(* Logix 5000 project; controller reports 1756-L63 rev 20.11; software revision 20.04; part 45 of 52 *)

        [132].log_data[58].valid := 1, [132].log_data[59].time := 3600.0, [132].log_data[59].valid := 1, [132].log_data[60].valid := 1, [132].log_data[61].valid := 1, [132].log_data[62].valid := 1, [132].log_data[63].valid := 1, [132].log_data[64].valid := 1, [132].log_data[65].valid := 1, [132].log_data[66].valid := 1, [132].log_data[67].valid := 1, [132].log_data[68].valid := 1, [132].log_data[69].valid := 1, [132].log_data[70].valid := 1, [132].log_data[71].valid := 1, [132].log_data[72].valid := 1, [132].log_data[73].valid := 1, [132].log_data[74].valid := 1, [132].log_data[75].valid := 1, [132].log_data[76].valid := 1, [132].log_data[77].valid := 1, [132].log_data[78].valid := 1, [132].log_data[79].valid := 1, [132].log_data[80].valid := 1, [132].log_data[81].valid := 1, [132].log_data[82].valid := 1, [132].log_data[83].valid := 1, [132].log_data[84].valid := 1, [132].log_data[85].valid := 1, [132].log_data[86].valid := 1, [132].log_data[87].valid := 1, [132].log_data[88].valid := 1, [132].log_data[89].valid := 1, [132].log_data[90].valid := 1, [132].log_data[91].valid := 1, [132].log_data[92].valid := 1, [132].log_data[93].valid := 1, [132].log_data[94].valid := 1, [132].log_data[95].valid := 1, [132].log_data[96].valid := 1, [132].log_data[97].valid := 1, [132].log_data[98].valid := 1, [132].log_data[99].valid := 1, [132].log_data[100].valid := 1, [132].log_data[101].valid := 1, [132].log_data[102].valid := 1, [132].log_data[103].valid := 1, [132].log_data[104].valid := 1, [132].log_data[105].valid := 1, [132].log_data[106].valid := 1, [132].log_data[107].valid := 1, [132].log_data[108].valid := 1, [132].log_data[109].valid := 1, [132].log_data[110].valid := 1, [132].log_data[111].valid := 1, [132].log_data[112].valid := 1, [132].log_data[113].valid := 1, [132].log_data[114].valid := 1, [132].log_data[115].valid := 1, [132].log_data[116].valid := 1,
        [132].log_data[117].valid := 1, [132].log_data[118].valid := 1, [132].log_data[119].valid := 1, [132].log_data[120].valid := 1, [132].log_data[121].valid := 1, [132].log_data[122].valid := 1, [132].log_data[123].valid := 1, [132].log_data[124].valid := 1, [132].time.Year := 2023, [132].time.Month := 1, [132].time.Day := 18, [132].time.Hour := 15, [132].time.Minute := 59, [132].time.Second := 59, [133].log_data[0].min := 1.0, [133].log_data[0].max := 1.0, [133].log_data[0].total := 3600.0, [133].log_data[0].time := 3600.0, [133].log_data[0].valid := 1, [133].log_data[1].max := 1.0, [133].log_data[1].total := 561.5, [133].log_data[1].time := 3600.0, [133].log_data[1].maxminute := 34, [133].log_data[1].valid := 1, [133].log_data[2].max := 1.0, [133].log_data[2].total := 558.0, [133].log_data[2].time := 3600.0, [133].log_data[2].maxminute := 34, [133].log_data[2].valid := 1, [133].log_data[3].time := 3600.0, [133].log_data[3].valid := 1, [133].log_data[4].time := 3600.0, [133].log_data[4].valid := 1, [133].log_data[5].max := 1.0, [133].log_data[5].total := 252.0, [133].log_data[5].time := 3600.0, [133].log_data[5].maxminute := 36, [133].log_data[5].valid := 1, [133].log_data[6].time := 3600.0, [133].log_data[6].valid := 1, [133].log_data[7].time := 3600.0, [133].log_data[7].valid := 1, [133].log_data[8].time := 3600.0, [133].log_data[8].valid := 1, [133].log_data[9].time := 3600.0, [133].log_data[9].valid := 1, [133].log_data[10].min := 1.0, [133].log_data[10].max := 1.0, [133].log_data[10].total := 3600.0, [133].log_data[10].time := 3600.0, [133].log_data[10].valid := 1, [133].log_data[11].time := 3600.0, [133].log_data[11].valid := 1, [133].log_data[12].min := 1.0, [133].log_data[12].max := 1.0, [133].log_data[12].total := 3600.0, [133].log_data[12].time := 3600.0, [133].log_data[12].valid := 1, [133].log_data[13].min := 1.0, [133].log_data[13].max := 1.0,
        [133].log_data[13].total := 3600.0, [133].log_data[13].time := 3600.0, [133].log_data[13].valid := 1, [133].log_data[14].time := 3600.0, [133].log_data[14].valid := 1, [133].log_data[15].time := 3600.0, [133].log_data[15].valid := 1, [133].log_data[16].time := 3600.0, [133].log_data[16].valid := 1, [133].log_data[17].min := 1.0, [133].log_data[17].max := 1.0, [133].log_data[17].total := 3600.0, [133].log_data[17].time := 3600.0, [133].log_data[17].valid := 1, [133].log_data[18].time := 3600.0, [133].log_data[18].valid := 1, [133].log_data[19].time := 3600.0, [133].log_data[19].valid := 1, [133].log_data[20].time := 3600.0, [133].log_data[20].valid := 1, [133].log_data[21].min := 1.0, [133].log_data[21].max := 1.0, [133].log_data[21].total := 3600.0, [133].log_data[21].time := 3600.0, [133].log_data[21].valid := 1, [133].log_data[22].time := 3600.0, [133].log_data[22].valid := 1, [133].log_data[23].time := 3600.0, [133].log_data[23].valid := 1, [133].log_data[24].time := 3600.0, [133].log_data[24].valid := 1, [133].log_data[25].time := 3600.0, [133].log_data[25].valid := 1, [133].log_data[26].time := 3600.0, [133].log_data[26].valid := 1, [133].log_data[27].time := 3600.0, [133].log_data[27].valid := 1, [133].log_data[28].time := 3600.0, [133].log_data[28].valid := 1, [133].log_data[29].min := 1.0, [133].log_data[29].max := 1.0, [133].log_data[29].total := 3600.0, [133].log_data[29].time := 3600.0, [133].log_data[29].valid := 1, [133].log_data[30].min := 1.0, [133].log_data[30].max := 1.0, [133].log_data[30].total := 3600.0, [133].log_data[30].time := 3600.0, [133].log_data[30].valid := 1, [133].log_data[31].time := 3600.0, [133].log_data[31].valid := 1, [133].log_data[32].time := 3600.0, [133].log_data[32].valid := 1, [133].log_data[33].time := 3600.0, [133].log_data[33].valid := 1, [133].log_data[34].time := 3600.0, [133].log_data[34].valid := 1, [133].log_data[35].time := 3600.0, [133].log_data[35].valid := 1, [133].log_data[36].time := 3600.0,
        [133].log_data[36].valid := 1, [133].log_data[37].max := 7.5544033, [133].log_data[37].total := 3699.229, [133].log_data[37].time := 3600.0, [133].log_data[37].maxminute := 36, [133].log_data[37].valid := 1, [133].log_data[38].time := 3600.0, [133].log_data[38].valid := 1, [133].log_data[39].min := 0.99541295, [133].log_data[39].max := 1.0215589, [133].log_data[39].total := 3606.4697, [133].log_data[39].time := 3600.0, [133].log_data[39].minminute := 45, [133].log_data[39].maxminute := 41, [133].log_data[39].valid := 1, [133].log_data[40].min := 7.5885, [133].log_data[40].max := 7.6244993, [133].log_data[40].total := 27393.127, [133].log_data[40].time := 3600.0, [133].log_data[40].minminute := 44, [133].log_data[40].maxminute := 51, [133].log_data[40].valid := 1, [133].log_data[41].min := 0.022343751, [133].log_data[41].max := 0.022932617, [133].log_data[41].total := 81.647255, [133].log_data[41].time := 3600.0, [133].log_data[41].minminute := 10, [133].log_data[41].valid := 1, [133].log_data[42].min := 2.291407, [133].log_data[42].max := 2.2958827, [133].log_data[42].total := 8257.927, [133].log_data[42].time := 3600.0, [133].log_data[42].minminute := 49, [133].log_data[42].maxminute := 6, [133].log_data[42].valid := 1, [133].log_data[43].min := -0.26000214, [133].log_data[43].max := -0.23999786, [133].log_data[43].total := -932.50854, [133].log_data[43].time := 3600.0, [133].log_data[43].valid := 1, [133].log_data[44].min := -0.30000305, [133].log_data[44].max := -0.27999878, [133].log_data[44].total := -1009.3977, [133].log_data[44].time := 3600.0, [133].log_data[44].valid := 1, [133].log_data[45].time := 3600.0, [133].log_data[45].valid := 1, [133].log_data[46].time := 3600.0, [133].log_data[46].valid := 1, [133].log_data[47].time := 3600.0, [133].log_data[47].valid := 1, [133].log_data[48].min := 6.7547326, [133].log_data[48].max := 6.977601, [133].log_data[48].total := 24541.125, [133].log_data[48].time := 3600.0, [133].log_data[48].maxminute := 43, [133].log_data[48].valid := 1, [133].log_data[49].min := 6.734528, [133].log_data[49].max := 9.605879, [133].log_data[49].total := 31908.559,
        [133].log_data[49].time := 3600.0, [133].log_data[49].minminute := 59, [133].log_data[49].maxminute := 37, [133].log_data[49].valid := 1, [133].log_data[50].min := 2.00227, [133].log_data[50].max := 2.1381822, [133].log_data[50].total := 7381.451, [133].log_data[50].time := 3600.0, [133].log_data[50].minminute := 11, [133].log_data[50].maxminute := 57, [133].log_data[50].valid := 1, [133].log_data[51].time := 3600.0, [133].log_data[51].valid := 1, [133].log_data[52].min := -1.6200027, [133].log_data[52].max := -1.4800034, [133].log_data[52].total := -5649.4478, [133].log_data[52].time := 3600.0, [133].log_data[52].minminute := 4, [133].log_data[52].maxminute := 31, [133].log_data[52].valid := 1, [133].log_data[53].min := -1.5800018, [133].log_data[53].max := -1.4599991, [133].log_data[53].total := -5378.804, [133].log_data[53].time := 3600.0, [133].log_data[53].minminute := 12, [133].log_data[53].maxminute := 1, [133].log_data[53].valid := 1, [133].log_data[54].time := 3600.0, [133].log_data[54].valid := 1, [133].log_data[55].time := 3600.0, [133].log_data[55].valid := 1, [133].log_data[56].min := 0.15898935, [133].log_data[56].max := 0.15938194, [133].log_data[56].total := 573.0084, [133].log_data[56].time := 3600.0, [133].log_data[56].minminute := 59, [133].log_data[56].maxminute := 7, [133].log_data[56].valid := 1, [133].log_data[57].min := 0.20103496, [133].log_data[57].max := 0.20142753, [133].log_data[57].total := 724.2275, [133].log_data[57].time := 3600.0, [133].log_data[57].minminute := 2, [133].log_data[57].maxminute := 41, [133].log_data[57].valid := 1, [133].log_data[58].time := 3600.0, [133].log_data[58].valid := 1, [133].log_data[59].time := 3600.0, [133].log_data[59].valid := 1, [133].log_data[60].valid := 1, [133].log_data[61].valid := 1, [133].log_data[62].valid := 1, [133].log_data[63].valid := 1, [133].log_data[64].valid := 1, [133].log_data[65].valid := 1, [133].log_data[66].valid := 1, [133].log_data[67].valid := 1, [133].log_data[68].valid := 1, [133].log_data[69].valid := 1, [133].log_data[70].valid := 1,
        [133].log_data[71].valid := 1, [133].log_data[72].valid := 1, [133].log_data[73].valid := 1, [133].log_data[74].valid := 1, [133].log_data[75].valid := 1, [133].log_data[76].valid := 1, [133].log_data[77].valid := 1, [133].log_data[78].valid := 1, [133].log_data[79].valid := 1, [133].log_data[80].valid := 1, [133].log_data[81].valid := 1, [133].log_data[82].valid := 1, [133].log_data[83].valid := 1, [133].log_data[84].valid := 1, [133].log_data[85].valid := 1, [133].log_data[86].valid := 1, [133].log_data[87].valid := 1, [133].log_data[88].valid := 1, [133].log_data[89].valid := 1, [133].log_data[90].valid := 1, [133].log_data[91].valid := 1, [133].log_data[92].valid := 1, [133].log_data[93].valid := 1, [133].log_data[94].valid := 1, [133].log_data[95].valid := 1, [133].log_data[96].valid := 1, [133].log_data[97].valid := 1, [133].log_data[98].valid := 1, [133].log_data[99].valid := 1, [133].log_data[100].valid := 1, [133].log_data[101].valid := 1, [133].log_data[102].valid := 1, [133].log_data[103].valid := 1, [133].log_data[104].valid := 1, [133].log_data[105].valid := 1, [133].log_data[106].valid := 1, [133].log_data[107].valid := 1, [133].log_data[108].valid := 1, [133].log_data[109].valid := 1, [133].log_data[110].valid := 1, [133].log_data[111].valid := 1, [133].log_data[112].valid := 1, [133].log_data[113].valid := 1, [133].log_data[114].valid := 1, [133].log_data[115].valid := 1, [133].log_data[116].valid := 1, [133].log_data[117].valid := 1, [133].log_data[118].valid := 1, [133].log_data[119].valid := 1, [133].log_data[120].valid := 1, [133].log_data[121].valid := 1, [133].log_data[122].valid := 1, [133].log_data[123].valid := 1, [133].log_data[124].valid := 1, [133].time.Year := 2023, [133].time.Month := 1, [133].time.Day := 18, [133].time.Hour := 16, [133].time.Minute := 59, [133].time.Second := 59,
        [134].log_data[0].min := 1.0, [134].log_data[0].max := 1.0, [134].log_data[0].total := 3600.0, [134].log_data[0].time := 3600.0, [134].log_data[0].valid := 1, [134].log_data[1].max := 1.0, [134].log_data[1].total := 524.749, [134].log_data[1].time := 3600.0, [134].log_data[1].maxminute := 51, [134].log_data[1].valid := 1, [134].log_data[2].max := 1.0, [134].log_data[2].total := 521.249, [134].log_data[2].time := 3600.0, [134].log_data[2].maxminute := 51, [134].log_data[2].valid := 1, [134].log_data[3].time := 3600.0, [134].log_data[3].valid := 1, [134].log_data[4].time := 3600.0, [134].log_data[4].valid := 1, [134].log_data[5].max := 1.0, [134].log_data[5].total := 224.249, [134].log_data[5].time := 3600.0, [134].log_data[5].maxminute := 53, [134].log_data[5].valid := 1, [134].log_data[6].time := 3600.0, [134].log_data[6].valid := 1, [134].log_data[7].time := 3600.0, [134].log_data[7].valid := 1, [134].log_data[8].max := 1.0, [134].log_data[8].total := 337.749, [134].log_data[8].time := 3600.0, [134].log_data[8].maxminute := 54, [134].log_data[8].valid := 1, [134].log_data[9].max := 1.0, [134].log_data[9].total := 334.249, [134].log_data[9].time := 3600.0, [134].log_data[9].maxminute := 54, [134].log_data[9].valid := 1, [134].log_data[10].min := 1.0, [134].log_data[10].max := 1.0, [134].log_data[10].total := 3600.0, [134].log_data[10].time := 3600.0, [134].log_data[10].valid := 1, [134].log_data[11].time := 3600.0, [134].log_data[11].valid := 1, [134].log_data[12].min := 1.0, [134].log_data[12].max := 1.0, [134].log_data[12].total := 3600.0, [134].log_data[12].time := 3600.0, [134].log_data[12].valid := 1, [134].log_data[13].min := 1.0, [134].log_data[13].max := 1.0, [134].log_data[13].total := 3600.0, [134].log_data[13].time := 3600.0, [134].log_data[13].valid := 1, [134].log_data[14].time := 3600.0, [134].log_data[14].valid := 1, [134].log_data[15].time := 3600.0, [134].log_data[15].valid := 1, [134].log_data[16].time := 3600.0,
        [134].log_data[16].valid := 1, [134].log_data[17].min := 1.0, [134].log_data[17].max := 1.0, [134].log_data[17].total := 3600.0, [134].log_data[17].time := 3600.0, [134].log_data[17].valid := 1, [134].log_data[18].time := 3600.0, [134].log_data[18].valid := 1, [134].log_data[19].time := 3600.0, [134].log_data[19].valid := 1, [134].log_data[20].time := 3600.0, [134].log_data[20].valid := 1, [134].log_data[21].min := 1.0, [134].log_data[21].max := 1.0, [134].log_data[21].total := 3600.0, [134].log_data[21].time := 3600.0, [134].log_data[21].valid := 1, [134].log_data[22].time := 3600.0, [134].log_data[22].valid := 1, [134].log_data[23].time := 3600.0, [134].log_data[23].valid := 1, [134].log_data[24].time := 3600.0, [134].log_data[24].valid := 1, [134].log_data[25].time := 3600.0, [134].log_data[25].valid := 1, [134].log_data[26].time := 3600.0, [134].log_data[26].valid := 1, [134].log_data[27].time := 3600.0, [134].log_data[27].valid := 1, [134].log_data[28].time := 3600.0, [134].log_data[28].valid := 1, [134].log_data[29].min := 1.0, [134].log_data[29].max := 1.0, [134].log_data[29].total := 3600.0, [134].log_data[29].time := 3600.0, [134].log_data[29].valid := 1, [134].log_data[30].min := 1.0, [134].log_data[30].max := 1.0, [134].log_data[30].total := 3600.0, [134].log_data[30].time := 3600.0, [134].log_data[30].valid := 1, [134].log_data[31].max := 1.0, [134].log_data[31].total := 57.249, [134].log_data[31].time := 3600.0, [134].log_data[31].maxminute := 54, [134].log_data[31].valid := 1, [134].log_data[32].max := 1.0, [134].log_data[32].total := 185.249, [134].log_data[32].time := 3600.0, [134].log_data[32].maxminute := 56, [134].log_data[32].valid := 1, [134].log_data[33].time := 3600.0, [134].log_data[33].valid := 1, [134].log_data[34].time := 3600.0, [134].log_data[34].valid := 1, [134].log_data[35].time := 3600.0, [134].log_data[35].valid := 1, [134].log_data[36].max := 1.0, [134].log_data[36].total := 327.249, [134].log_data[36].time := 3600.0,
        [134].log_data[36].maxminute := 54, [134].log_data[36].valid := 1, [134].log_data[37].max := 9.523992, [134].log_data[37].total := 3687.952, [134].log_data[37].time := 3600.0, [134].log_data[37].maxminute := 53, [134].log_data[37].valid := 1, [134].log_data[38].time := 3600.0, [134].log_data[38].valid := 1, [134].log_data[39].min := 0.99423516, [134].log_data[39].max := 1.0213233, [134].log_data[39].total := 3603.442, [134].log_data[39].time := 3600.0, [134].log_data[39].minminute := 13, [134].log_data[39].maxminute := 58, [134].log_data[39].valid := 1, [134].log_data[40].min := 7.592622, [134].log_data[40].max := 7.6244993, [134].log_data[40].total := 27393.01, [134].log_data[40].time := 3600.0, [134].log_data[40].minminute := 1, [134].log_data[40].maxminute := 10, [134].log_data[40].valid := 1, [134].log_data[41].min := 0.022343751, [134].log_data[41].max := 0.022932617, [134].log_data[41].total := 81.438286, [134].log_data[41].time := 3600.0, [134].log_data[41].minminute := 1, [134].log_data[41].maxminute := 15, [134].log_data[41].valid := 1, [134].log_data[42].min := 2.2912893, [134].log_data[42].max := 2.296118, [134].log_data[42].total := 8257.677, [134].log_data[42].time := 3600.0, [134].log_data[42].minminute := 38, [134].log_data[42].maxminute := 18, [134].log_data[42].valid := 1, [134].log_data[43].min := -0.26000214, [134].log_data[43].max := -0.23999786, [134].log_data[43].total := -926.4218, [134].log_data[43].time := 3600.0, [134].log_data[43].maxminute := 1, [134].log_data[43].valid := 1, [134].log_data[44].min := -0.30000305, [134].log_data[44].max := -0.27999878, [134].log_data[44].total := -1008.3122, [134].log_data[44].time := 3600.0, [134].log_data[44].valid := 1, [134].log_data[45].time := 3600.0, [134].log_data[45].valid := 1, [134].log_data[46].time := 3600.0, [134].log_data[46].valid := 1, [134].log_data[47].time := 3600.0, [134].log_data[47].valid := 1, [134].log_data[48].min := 6.618977, [134].log_data[48].max := 6.854762, [134].log_data[48].total := 24051.516, [134].log_data[48].time := 3600.0, [134].log_data[48].minminute := 28, [134].log_data[48].maxminute := 59,
        [134].log_data[48].valid := 1, [134].log_data[49].min := 6.092655, [134].log_data[49].max := 8.969305, [134].log_data[49].total := 25809.742, [134].log_data[49].time := 3600.0, [134].log_data[49].minminute := 16, [134].log_data[49].maxminute := 54, [134].log_data[49].valid := 1, [134].log_data[50].min := 2.0787058, [134].log_data[50].max := 2.1524327, [134].log_data[50].total := 7686.3364, [134].log_data[50].time := 3600.0, [134].log_data[50].minminute := 58, [134].log_data[50].maxminute := 54, [134].log_data[50].valid := 1, [134].log_data[51].time := 3600.0, [134].log_data[51].valid := 1, [134].log_data[52].min := -4.119995, [134].log_data[52].max := 0.13999939, [134].log_data[52].total := -5775.382, [134].log_data[52].time := 3600.0, [134].log_data[52].minminute := 54, [134].log_data[52].maxminute := 56, [134].log_data[52].valid := 1, [134].log_data[53].min := -4.079994, [134].log_data[53].max := -1.4599991, [134].log_data[53].total := -5722.698, [134].log_data[53].time := 3600.0, [134].log_data[53].minminute := 54, [134].log_data[53].valid := 1, [134].log_data[54].max := 0.513, [134].log_data[54].total := 92.831985, [134].log_data[54].time := 3600.0, [134].log_data[54].maxminute := 57, [134].log_data[54].valid := 1, [134].log_data[55].max := 0.526, [134].log_data[55].total := 128.63133, [134].log_data[55].time := 3600.0, [134].log_data[55].maxminute := 54, [134].log_data[55].valid := 1, [134].log_data[56].min := 0.15898935, [134].log_data[56].max := 0.15942119, [134].log_data[56].total := 572.9697, [134].log_data[56].time := 3600.0, [134].log_data[56].minminute := 45, [134].log_data[56].maxminute := 38, [134].log_data[56].valid := 1, [134].log_data[57].min := 0.20103496, [134].log_data[57].max := 0.20142753, [134].log_data[57].total := 724.2705, [134].log_data[57].time := 3600.0, [134].log_data[57].maxminute := 36, [134].log_data[57].valid := 1, [134].log_data[58].time := 3600.0, [134].log_data[58].valid := 1, [134].log_data[59].time := 3600.0, [134].log_data[59].valid := 1, [134].log_data[60].valid := 1, [134].log_data[61].valid := 1, [134].log_data[62].valid := 1,
        [134].log_data[63].valid := 1, [134].log_data[64].valid := 1, [134].log_data[65].valid := 1, [134].log_data[66].valid := 1, [134].log_data[67].valid := 1, [134].log_data[68].valid := 1, [134].log_data[69].valid := 1, [134].log_data[70].valid := 1, [134].log_data[71].valid := 1, [134].log_data[72].valid := 1, [134].log_data[73].valid := 1, [134].log_data[74].valid := 1, [134].log_data[75].valid := 1, [134].log_data[76].valid := 1, [134].log_data[77].valid := 1, [134].log_data[78].valid := 1, [134].log_data[79].valid := 1, [134].log_data[80].valid := 1, [134].log_data[81].valid := 1, [134].log_data[82].valid := 1, [134].log_data[83].valid := 1, [134].log_data[84].valid := 1, [134].log_data[85].valid := 1, [134].log_data[86].valid := 1, [134].log_data[87].valid := 1, [134].log_data[88].valid := 1, [134].log_data[89].valid := 1, [134].log_data[90].valid := 1, [134].log_data[91].valid := 1, [134].log_data[92].valid := 1, [134].log_data[93].valid := 1, [134].log_data[94].valid := 1, [134].log_data[95].valid := 1, [134].log_data[96].valid := 1, [134].log_data[97].valid := 1, [134].log_data[98].valid := 1, [134].log_data[99].valid := 1, [134].log_data[100].valid := 1, [134].log_data[101].valid := 1, [134].log_data[102].valid := 1, [134].log_data[103].valid := 1, [134].log_data[104].valid := 1, [134].log_data[105].valid := 1, [134].log_data[106].valid := 1, [134].log_data[107].valid := 1, [134].log_data[108].valid := 1, [134].log_data[109].valid := 1, [134].log_data[110].valid := 1, [134].log_data[111].valid := 1, [134].log_data[112].valid := 1, [134].log_data[113].valid := 1, [134].log_data[114].valid := 1, [134].log_data[115].valid := 1, [134].log_data[116].valid := 1, [134].log_data[117].valid := 1, [134].log_data[118].valid := 1, [134].log_data[119].valid := 1, [134].log_data[120].valid := 1, [134].log_data[121].valid := 1, [134].log_data[122].valid := 1,
        [134].log_data[123].valid := 1, [134].log_data[124].valid := 1, [134].time.Year := 2023, [134].time.Month := 1, [134].time.Day := 18, [134].time.Hour := 17, [134].time.Minute := 59, [134].time.Second := 59, [135].log_data[0].min := 1.0, [135].log_data[0].max := 1.0, [135].log_data[0].total := 3600.0, [135].log_data[0].time := 3600.0, [135].log_data[0].valid := 1, [135].log_data[1].max := 1.0, [135].log_data[1].total := 41.751, [135].log_data[1].time := 3600.0, [135].log_data[1].valid := 1, [135].log_data[2].max := 1.0, [135].log_data[2].total := 41.751, [135].log_data[2].time := 3600.0, [135].log_data[2].valid := 1, [135].log_data[3].time := 3600.0, [135].log_data[3].valid := 1, [135].log_data[4].time := 3600.0, [135].log_data[4].valid := 1, [135].log_data[5].max := 1.0, [135].log_data[5].total := 18.751, [135].log_data[5].time := 3600.0, [135].log_data[5].valid := 1, [135].log_data[6].time := 3600.0, [135].log_data[6].valid := 1, [135].log_data[7].time := 3600.0, [135].log_data[7].valid := 1, [135].log_data[8].min := 1.0, [135].log_data[8].max := 1.0, [135].log_data[8].total := 3600.0, [135].log_data[8].time := 3600.0, [135].log_data[8].valid := 1, [135].log_data[9].min := 1.0, [135].log_data[9].max := 1.0, [135].log_data[9].total := 3600.0, [135].log_data[9].time := 3600.0, [135].log_data[9].valid := 1, [135].log_data[10].min := 1.0, [135].log_data[10].max := 1.0, [135].log_data[10].total := 3600.0, [135].log_data[10].time := 3600.0, [135].log_data[10].valid := 1, [135].log_data[11].time := 3600.0, [135].log_data[11].valid := 1, [135].log_data[12].min := 1.0, [135].log_data[12].max := 1.0, [135].log_data[12].total := 3600.0, [135].log_data[12].time := 3600.0, [135].log_data[12].valid := 1, [135].log_data[13].min := 1.0, [135].log_data[13].max := 1.0, [135].log_data[13].total := 3600.0, [135].log_data[13].time := 3600.0, [135].log_data[13].valid := 1,
        [135].log_data[14].time := 3600.0, [135].log_data[14].valid := 1, [135].log_data[15].time := 3600.0, [135].log_data[15].valid := 1, [135].log_data[16].time := 3600.0, [135].log_data[16].valid := 1, [135].log_data[17].min := 1.0, [135].log_data[17].max := 1.0, [135].log_data[17].total := 3600.0, [135].log_data[17].time := 3600.0, [135].log_data[17].valid := 1, [135].log_data[18].time := 3600.0, [135].log_data[18].valid := 1, [135].log_data[19].time := 3600.0, [135].log_data[19].valid := 1, [135].log_data[20].time := 3600.0, [135].log_data[20].valid := 1, [135].log_data[21].min := 1.0, [135].log_data[21].max := 1.0, [135].log_data[21].total := 3600.0, [135].log_data[21].time := 3600.0, [135].log_data[21].valid := 1, [135].log_data[22].time := 3600.0, [135].log_data[22].valid := 1, [135].log_data[23].time := 3600.0, [135].log_data[23].valid := 1, [135].log_data[24].time := 3600.0, [135].log_data[24].valid := 1, [135].log_data[25].time := 3600.0, [135].log_data[25].valid := 1, [135].log_data[26].time := 3600.0, [135].log_data[26].valid := 1, [135].log_data[27].time := 3600.0, [135].log_data[27].valid := 1, [135].log_data[28].time := 3600.0, [135].log_data[28].valid := 1, [135].log_data[29].min := 1.0, [135].log_data[29].max := 1.0, [135].log_data[29].total := 3600.0, [135].log_data[29].time := 3600.0, [135].log_data[29].valid := 1, [135].log_data[30].min := 1.0, [135].log_data[30].max := 1.0, [135].log_data[30].total := 3600.0, [135].log_data[30].time := 3600.0, [135].log_data[30].valid := 1, [135].log_data[31].max := 1.0, [135].log_data[31].total := 1629.998, [135].log_data[31].time := 3600.0, [135].log_data[31].maxminute := 7, [135].log_data[31].valid := 1, [135].log_data[32].max := 1.0, [135].log_data[32].total := 1444.498, [135].log_data[32].time := 3600.0, [135].log_data[32].minminute := 5, [135].log_data[32].valid := 1, [135].log_data[33].time := 3600.0, [135].log_data[33].valid := 1, [135].log_data[34].time := 3600.0, [135].log_data[34].valid := 1,
        [135].log_data[35].max := 1.0, [135].log_data[35].total := 1629.498, [135].log_data[35].time := 3600.0, [135].log_data[35].maxminute := 2, [135].log_data[35].valid := 1, [135].log_data[36].max := 1.0, [135].log_data[36].total := 1440.998, [135].log_data[36].time := 3600.0, [135].log_data[36].minminute := 1, [135].log_data[36].valid := 1, [135].log_data[37].time := 3600.0, [135].log_data[37].valid := 1, [135].log_data[38].time := 3600.0, [135].log_data[38].valid := 1, [135].log_data[39].min := 0.99623734, [135].log_data[39].max := 1.0076615, [135].log_data[39].total := 3603.6245, [135].log_data[39].time := 3600.0, [135].log_data[39].minminute := 43, [135].log_data[39].valid := 1, [135].log_data[40].min := 7.586851, [135].log_data[40].max := 7.620378, [135].log_data[40].total := 27389.994, [135].log_data[40].time := 3600.0, [135].log_data[40].minminute := 28, [135].log_data[40].maxminute := 40, [135].log_data[40].valid := 1, [135].log_data[41].min := 0.022343751, [135].log_data[41].max := 0.022932617, [135].log_data[41].total := 81.52236, [135].log_data[41].time := 3600.0, [135].log_data[41].minminute := 4, [135].log_data[41].maxminute := 13, [135].log_data[41].valid := 1, [135].log_data[42].min := 2.290936, [135].log_data[42].max := 2.2957647, [135].log_data[42].total := 8257.714, [135].log_data[42].time := 3600.0, [135].log_data[42].minminute := 10, [135].log_data[42].maxminute := 5, [135].log_data[42].valid := 1, [135].log_data[43].min := -0.26000214, [135].log_data[43].max := -0.23999786, [135].log_data[43].total := -934.87366, [135].log_data[43].time := 3600.0, [135].log_data[43].valid := 1, [135].log_data[44].min := -0.30000305, [135].log_data[44].max := -0.27999878, [135].log_data[44].total := -1016.6125, [135].log_data[44].time := 3600.0, [135].log_data[44].valid := 1, [135].log_data[45].time := 3600.0, [135].log_data[45].valid := 1, [135].log_data[46].time := 3600.0, [135].log_data[46].valid := 1, [135].log_data[47].time := 3600.0, [135].log_data[47].valid := 1, [135].log_data[48].min := 6.677511, [135].log_data[48].max := 6.8819685, [135].log_data[48].total := 24228.434,
        [135].log_data[48].time := 3600.0, [135].log_data[48].minminute := 26, [135].log_data[48].valid := 1, [135].log_data[49].min := 6.88842, [135].log_data[49].max := 9.422542, [135].log_data[49].total := 28967.625, [135].log_data[49].time := 3600.0, [135].log_data[49].minminute := 21, [135].log_data[49].maxminute := 59, [135].log_data[49].valid := 1, [135].log_data[50].min := 2.059273, [135].log_data[50].max := 2.1438353, [135].log_data[50].total := 7571.9165, [135].log_data[50].time := 3600.0, [135].log_data[50].minminute := 59, [135].log_data[50].valid := 1, [135].log_data[51].time := 3600.0, [135].log_data[51].valid := 1, [135].log_data[52].min := -2.7600021, [135].log_data[52].max := 0.13999939, [135].log_data[52].total := -7516.524, [135].log_data[52].time := 3600.0, [135].log_data[52].minminute := 39, [135].log_data[52].maxminute := 6, [135].log_data[52].valid := 1, [135].log_data[53].min := -2.4400024, [135].log_data[53].max := 0.3600006, [135].log_data[53].total := -6614.5444, [135].log_data[53].time := 3600.0, [135].log_data[53].minminute := 46, [135].log_data[53].maxminute := 12, [135].log_data[53].valid := 1, [135].log_data[54].max := 0.5195, [135].log_data[54].total := 1221.1208, [135].log_data[54].time := 3600.0, [135].log_data[54].minminute := 5, [135].log_data[54].maxminute := 49, [135].log_data[54].valid := 1, [135].log_data[55].max := 0.557, [135].log_data[55].total := 1217.2502, [135].log_data[55].time := 3600.0, [135].log_data[55].minminute := 1, [135].log_data[55].maxminute := 2, [135].log_data[55].valid := 1, [135].log_data[56].min := 0.15898935, [135].log_data[56].max := 0.15938194, [135].log_data[56].total := 572.84296, [135].log_data[56].time := 3600.0, [135].log_data[56].minminute := 9, [135].log_data[56].maxminute := 37, [135].log_data[56].valid := 1, [135].log_data[57].min := 0.20095645, [135].log_data[57].max := 0.20138828, [135].log_data[57].total := 724.062, [135].log_data[57].time := 3600.0, [135].log_data[57].minminute := 19, [135].log_data[57].maxminute := 3, [135].log_data[57].valid := 1, [135].log_data[58].time := 3600.0, [135].log_data[58].valid := 1,
        [135].log_data[59].time := 3600.0, [135].log_data[59].valid := 1, [135].log_data[60].valid := 1, [135].log_data[61].valid := 1, [135].log_data[62].valid := 1, [135].log_data[63].valid := 1, [135].log_data[64].valid := 1, [135].log_data[65].valid := 1, [135].log_data[66].valid := 1, [135].log_data[67].valid := 1, [135].log_data[68].valid := 1, [135].log_data[69].valid := 1, [135].log_data[70].valid := 1, [135].log_data[71].valid := 1, [135].log_data[72].valid := 1, [135].log_data[73].valid := 1, [135].log_data[74].valid := 1, [135].log_data[75].valid := 1, [135].log_data[76].valid := 1, [135].log_data[77].valid := 1, [135].log_data[78].valid := 1, [135].log_data[79].valid := 1, [135].log_data[80].valid := 1, [135].log_data[81].valid := 1, [135].log_data[82].valid := 1, [135].log_data[83].valid := 1, [135].log_data[84].valid := 1, [135].log_data[85].valid := 1, [135].log_data[86].valid := 1, [135].log_data[87].valid := 1, [135].log_data[88].valid := 1, [135].log_data[89].valid := 1, [135].log_data[90].valid := 1, [135].log_data[91].valid := 1, [135].log_data[92].valid := 1, [135].log_data[93].valid := 1, [135].log_data[94].valid := 1, [135].log_data[95].valid := 1, [135].log_data[96].valid := 1, [135].log_data[97].valid := 1, [135].log_data[98].valid := 1, [135].log_data[99].valid := 1, [135].log_data[100].valid := 1, [135].log_data[101].valid := 1, [135].log_data[102].valid := 1, [135].log_data[103].valid := 1, [135].log_data[104].valid := 1, [135].log_data[105].valid := 1, [135].log_data[106].valid := 1, [135].log_data[107].valid := 1, [135].log_data[108].valid := 1, [135].log_data[109].valid := 1, [135].log_data[110].valid := 1, [135].log_data[111].valid := 1, [135].log_data[112].valid := 1, [135].log_data[113].valid := 1, [135].log_data[114].valid := 1, [135].log_data[115].valid := 1, [135].log_data[116].valid := 1, [135].log_data[117].valid := 1,
        [135].log_data[118].valid := 1, [135].log_data[119].valid := 1, [135].log_data[120].valid := 1, [135].log_data[121].valid := 1, [135].log_data[122].valid := 1, [135].log_data[123].valid := 1, [135].log_data[124].valid := 1, [135].time.Year := 2023, [135].time.Month := 1, [135].time.Day := 18, [135].time.Hour := 18, [135].time.Minute := 59, [135].time.Second := 59, [136].log_data[0].min := 1.0, [136].log_data[0].max := 1.0, [136].log_data[0].total := 3600.0, [136].log_data[0].time := 3600.0, [136].log_data[0].valid := 1, [136].log_data[1].max := 1.0, [136].log_data[1].total := 544.0, [136].log_data[1].time := 3600.0, [136].log_data[1].maxminute := 22, [136].log_data[1].valid := 1, [136].log_data[2].max := 1.0, [136].log_data[2].total := 540.5, [136].log_data[2].time := 3600.0, [136].log_data[2].maxminute := 22, [136].log_data[2].valid := 1, [136].log_data[3].time := 3600.0, [136].log_data[3].valid := 1, [136].log_data[4].time := 3600.0, [136].log_data[4].valid := 1, [136].log_data[5].max := 1.0, [136].log_data[5].total := 246.0, [136].log_data[5].time := 3600.0, [136].log_data[5].maxminute := 25, [136].log_data[5].valid := 1, [136].log_data[6].time := 3600.0, [136].log_data[6].valid := 1, [136].log_data[7].time := 3600.0, [136].log_data[7].valid := 1, [136].log_data[8].min := 1.0, [136].log_data[8].max := 1.0, [136].log_data[8].total := 3600.0, [136].log_data[8].time := 3600.0, [136].log_data[8].valid := 1, [136].log_data[9].min := 1.0, [136].log_data[9].max := 1.0, [136].log_data[9].total := 3600.0, [136].log_data[9].time := 3600.0, [136].log_data[9].valid := 1, [136].log_data[10].min := 1.0, [136].log_data[10].max := 1.0, [136].log_data[10].total := 3600.0, [136].log_data[10].time := 3600.0, [136].log_data[10].valid := 1, [136].log_data[11].time := 3600.0, [136].log_data[11].valid := 1, [136].log_data[12].min := 1.0, [136].log_data[12].max := 1.0,
        [136].log_data[12].total := 3600.0, [136].log_data[12].time := 3600.0, [136].log_data[12].valid := 1, [136].log_data[13].min := 1.0, [136].log_data[13].max := 1.0, [136].log_data[13].total := 3600.0, [136].log_data[13].time := 3600.0, [136].log_data[13].valid := 1, [136].log_data[14].time := 3600.0, [136].log_data[14].valid := 1, [136].log_data[15].time := 3600.0, [136].log_data[15].valid := 1, [136].log_data[16].time := 3600.0, [136].log_data[16].valid := 1, [136].log_data[17].min := 1.0, [136].log_data[17].max := 1.0, [136].log_data[17].total := 3600.0, [136].log_data[17].time := 3600.0, [136].log_data[17].valid := 1, [136].log_data[18].time := 3600.0, [136].log_data[18].valid := 1, [136].log_data[19].time := 3600.0, [136].log_data[19].valid := 1, [136].log_data[20].time := 3600.0, [136].log_data[20].valid := 1, [136].log_data[21].min := 1.0, [136].log_data[21].max := 1.0, [136].log_data[21].total := 3600.0, [136].log_data[21].time := 3600.0, [136].log_data[21].valid := 1, [136].log_data[22].time := 3600.0, [136].log_data[22].valid := 1, [136].log_data[23].time := 3600.0, [136].log_data[23].valid := 1, [136].log_data[24].time := 3600.0, [136].log_data[24].valid := 1, [136].log_data[25].time := 3600.0, [136].log_data[25].valid := 1, [136].log_data[26].time := 3600.0, [136].log_data[26].valid := 1, [136].log_data[27].time := 3600.0, [136].log_data[27].valid := 1, [136].log_data[28].time := 3600.0, [136].log_data[28].valid := 1, [136].log_data[29].min := 1.0, [136].log_data[29].max := 1.0, [136].log_data[29].total := 3600.0, [136].log_data[29].time := 3600.0, [136].log_data[29].valid := 1, [136].log_data[30].min := 1.0, [136].log_data[30].max := 1.0, [136].log_data[30].total := 3600.0, [136].log_data[30].time := 3600.0, [136].log_data[30].valid := 1, [136].log_data[31].max := 1.0, [136].log_data[31].total := 1524.7471, [136].log_data[31].time := 3600.0, [136].log_data[31].maxminute := 10, [136].log_data[31].valid := 1, [136].log_data[32].max := 1.0,
        [136].log_data[32].total := 1629.998, [136].log_data[32].time := 3600.0, [136].log_data[32].valid := 1, [136].log_data[33].time := 3600.0, [136].log_data[33].valid := 1, [136].log_data[34].time := 3600.0, [136].log_data[34].valid := 1, [136].log_data[35].max := 1.0, [136].log_data[35].total := 1629.7471, [136].log_data[35].time := 3600.0, [136].log_data[35].maxminute := 5, [136].log_data[35].valid := 1, [136].log_data[36].max := 1.0, [136].log_data[36].total := 1440.7471, [136].log_data[36].time := 3600.0, [136].log_data[36].minminute := 4, [136].log_data[36].valid := 1, [136].log_data[37].max := 7.557152, [136].log_data[37].total := 3566.1763, [136].log_data[37].time := 3600.0, [136].log_data[37].maxminute := 24, [136].log_data[37].valid := 1, [136].log_data[38].time := 3600.0, [136].log_data[38].valid := 1, [136].log_data[39].min := 0.9938818, [136].log_data[39].max := 1.0219122, [136].log_data[39].total := 3606.7239, [136].log_data[39].time := 3600.0, [136].log_data[39].minminute := 55, [136].log_data[39].maxminute := 29, [136].log_data[39].valid := 1, [136].log_data[40].min := 7.6000414, [136].log_data[40].max := 7.6162558, [136].log_data[40].total := 27396.957, [136].log_data[40].time := 3600.0, [136].log_data[40].minminute := 17, [136].log_data[40].valid := 1, [136].log_data[41].min := 0.022540038, [136].log_data[41].max := 0.022932617, [136].log_data[41].total := 81.802284, [136].log_data[41].time := 3600.0, [136].log_data[41].maxminute := 1, [136].log_data[41].valid := 1, [136].log_data[42].min := 2.290936, [136].log_data[42].max := 2.2958827, [136].log_data[42].total := 8257.7, [136].log_data[42].time := 3600.0, [136].log_data[42].minminute := 25, [136].log_data[42].maxminute := 12, [136].log_data[42].valid := 1, [136].log_data[43].min := -0.27999878, [136].log_data[43].max := -0.26000214, [136].log_data[43].total := -936.8631, [136].log_data[43].time := 3600.0, [136].log_data[43].minminute := 31, [136].log_data[43].valid := 1, [136].log_data[44].min := -0.30000305, [136].log_data[44].max := -0.27999878, [136].log_data[44].total := -1075.9814, [136].log_data[44].time := 3600.0,
        [136].log_data[44].valid := 1, [136].log_data[45].time := 3600.0, [136].log_data[45].valid := 1, [136].log_data[46].time := 3600.0, [136].log_data[46].valid := 1, [136].log_data[47].time := 3600.0, [136].log_data[47].valid := 1, [136].log_data[48].min := 6.6148553, [136].log_data[48].max := 6.9306097, [136].log_data[48].total := 24285.6, [136].log_data[48].time := 3600.0, [136].log_data[48].minminute := 56, [136].log_data[48].maxminute := 32, [136].log_data[48].valid := 1, [136].log_data[49].min := 6.7529798, [136].log_data[49].max := 9.563283, [136].log_data[49].total := 30213.775, [136].log_data[49].time := 3600.0, [136].log_data[49].minminute := 52, [136].log_data[49].maxminute := 25, [136].log_data[49].valid := 1, [136].log_data[50].min := 2.0217028, [136].log_data[50].max := 2.141362, [136].log_data[50].total := 7507.11, [136].log_data[50].time := 3600.0, [136].log_data[50].minminute := 25, [136].log_data[50].maxminute := 31, [136].log_data[50].valid := 1, [136].log_data[51].time := 3600.0, [136].log_data[51].valid := 1, [136].log_data[52].min := -2.7600021, [136].log_data[52].max := 0.11999512, [136].log_data[52].total := -7773.9062, [136].log_data[52].time := 3600.0, [136].log_data[52].minminute := 10, [136].log_data[52].valid := 1, [136].log_data[53].min := -2.4400024, [136].log_data[53].max := 0.30000305, [136].log_data[53].total := -6738.13, [136].log_data[53].time := 3600.0, [136].log_data[53].minminute := 5, [136].log_data[53].maxminute := 5, [136].log_data[53].valid := 1, [136].log_data[54].max := 0.532, [136].log_data[54].total := 1249.9996, [136].log_data[54].time := 3600.0, [136].log_data[54].maxminute := 52, [136].log_data[54].valid := 1, [136].log_data[55].max := 0.52900004, [136].log_data[55].total := 1216.8845, [136].log_data[55].time := 3600.0, [136].log_data[55].minminute := 4, [136].log_data[55].maxminute := 5, [136].log_data[55].valid := 1, [136].log_data[56].min := 0.15898935, [136].log_data[56].max := 0.15942119, [136].log_data[56].total := 573.08276, [136].log_data[56].time := 3600.0, [136].log_data[56].minminute := 6, [136].log_data[56].maxminute := 16,
        [136].log_data[56].valid := 1, [136].log_data[57].min := 0.20087793, [136].log_data[57].max := 0.20134902, [136].log_data[57].total := 723.77484, [136].log_data[57].time := 3600.0, [136].log_data[57].minminute := 20, [136].log_data[57].maxminute := 1, [136].log_data[57].valid := 1, [136].log_data[58].time := 3600.0, [136].log_data[58].valid := 1, [136].log_data[59].time := 3600.0, [136].log_data[59].valid := 1, [136].log_data[60].valid := 1, [136].log_data[61].valid := 1, [136].log_data[62].valid := 1, [136].log_data[63].valid := 1, [136].log_data[64].valid := 1, [136].log_data[65].valid := 1, [136].log_data[66].valid := 1, [136].log_data[67].valid := 1, [136].log_data[68].valid := 1, [136].log_data[69].valid := 1, [136].log_data[70].valid := 1, [136].log_data[71].valid := 1, [136].log_data[72].valid := 1, [136].log_data[73].valid := 1, [136].log_data[74].valid := 1, [136].log_data[75].valid := 1, [136].log_data[76].valid := 1, [136].log_data[77].valid := 1, [136].log_data[78].valid := 1, [136].log_data[79].valid := 1, [136].log_data[80].valid := 1, [136].log_data[81].valid := 1, [136].log_data[82].valid := 1, [136].log_data[83].valid := 1, [136].log_data[84].valid := 1, [136].log_data[85].valid := 1, [136].log_data[86].valid := 1, [136].log_data[87].valid := 1, [136].log_data[88].valid := 1, [136].log_data[89].valid := 1, [136].log_data[90].valid := 1, [136].log_data[91].valid := 1, [136].log_data[92].valid := 1, [136].log_data[93].valid := 1, [136].log_data[94].valid := 1, [136].log_data[95].valid := 1, [136].log_data[96].valid := 1, [136].log_data[97].valid := 1, [136].log_data[98].valid := 1, [136].log_data[99].valid := 1, [136].log_data[100].valid := 1, [136].log_data[101].valid := 1, [136].log_data[102].valid := 1, [136].log_data[103].valid := 1, [136].log_data[104].valid := 1, [136].log_data[105].valid := 1, [136].log_data[106].valid := 1, [136].log_data[107].valid := 1,
        [136].log_data[108].valid := 1, [136].log_data[109].valid := 1, [136].log_data[110].valid := 1, [136].log_data[111].valid := 1, [136].log_data[112].valid := 1, [136].log_data[113].valid := 1, [136].log_data[114].valid := 1, [136].log_data[115].valid := 1, [136].log_data[116].valid := 1, [136].log_data[117].valid := 1, [136].log_data[118].valid := 1, [136].log_data[119].valid := 1, [136].log_data[120].valid := 1, [136].log_data[121].valid := 1, [136].log_data[122].valid := 1, [136].log_data[123].valid := 1, [136].log_data[124].valid := 1, [136].time.Year := 2023, [136].time.Month := 1, [136].time.Day := 18, [136].time.Hour := 19, [136].time.Minute := 59, [136].time.Second := 59, [137].log_data[0].min := 1.0, [137].log_data[0].max := 1.0, [137].log_data[0].total := 3600.0, [137].log_data[0].time := 3600.0, [137].log_data[0].valid := 1, [137].log_data[1].max := 1.0, [137].log_data[1].total := 587.0, [137].log_data[1].time := 3600.0, [137].log_data[1].maxminute := 32, [137].log_data[1].valid := 1, [137].log_data[2].max := 1.0, [137].log_data[2].total := 583.5, [137].log_data[2].time := 3600.0, [137].log_data[2].maxminute := 32, [137].log_data[2].valid := 1, [137].log_data[3].time := 3600.0, [137].log_data[3].valid := 1, [137].log_data[4].time := 3600.0, [137].log_data[4].valid := 1, [137].log_data[5].max := 1.0, [137].log_data[5].total := 244.5, [137].log_data[5].time := 3600.0, [137].log_data[5].maxminute := 35, [137].log_data[5].valid := 1, [137].log_data[6].time := 3600.0, [137].log_data[6].valid := 1, [137].log_data[7].time := 3600.0, [137].log_data[7].valid := 1, [137].log_data[8].min := 1.0, [137].log_data[8].max := 1.0, [137].log_data[8].total := 3600.0, [137].log_data[8].time := 3600.0, [137].log_data[8].valid := 1, [137].log_data[9].min := 1.0, [137].log_data[9].max := 1.0, [137].log_data[9].total := 3600.0, [137].log_data[9].time := 3600.0,
        [137].log_data[9].valid := 1, [137].log_data[10].min := 1.0, [137].log_data[10].max := 1.0, [137].log_data[10].total := 3600.0, [137].log_data[10].time := 3600.0, [137].log_data[10].valid := 1, [137].log_data[11].time := 3600.0, [137].log_data[11].valid := 1, [137].log_data[12].min := 1.0, [137].log_data[12].max := 1.0, [137].log_data[12].total := 3600.0, [137].log_data[12].time := 3600.0, [137].log_data[12].valid := 1, [137].log_data[13].min := 1.0, [137].log_data[13].max := 1.0, [137].log_data[13].total := 3600.0, [137].log_data[13].time := 3600.0, [137].log_data[13].valid := 1, [137].log_data[14].time := 3600.0, [137].log_data[14].valid := 1, [137].log_data[15].time := 3600.0, [137].log_data[15].valid := 1, [137].log_data[16].time := 3600.0, [137].log_data[16].valid := 1, [137].log_data[17].min := 1.0, [137].log_data[17].max := 1.0, [137].log_data[17].total := 3600.0, [137].log_data[17].time := 3600.0, [137].log_data[17].valid := 1, [137].log_data[18].time := 3600.0, [137].log_data[18].valid := 1, [137].log_data[19].time := 3600.0, [137].log_data[19].valid := 1, [137].log_data[20].time := 3600.0, [137].log_data[20].valid := 1, [137].log_data[21].min := 1.0, [137].log_data[21].max := 1.0, [137].log_data[21].total := 3600.0, [137].log_data[21].time := 3600.0, [137].log_data[21].valid := 1, [137].log_data[22].time := 3600.0, [137].log_data[22].valid := 1, [137].log_data[23].time := 3600.0, [137].log_data[23].valid := 1, [137].log_data[24].time := 3600.0, [137].log_data[24].valid := 1, [137].log_data[25].time := 3600.0, [137].log_data[25].valid := 1, [137].log_data[26].time := 3600.0, [137].log_data[26].valid := 1, [137].log_data[27].time := 3600.0, [137].log_data[27].valid := 1, [137].log_data[28].time := 3600.0, [137].log_data[28].valid := 1, [137].log_data[29].min := 1.0, [137].log_data[29].max := 1.0, [137].log_data[29].total := 3600.0, [137].log_data[29].time := 3600.0, [137].log_data[29].valid := 1, [137].log_data[30].min := 1.0,
        [137].log_data[30].max := 1.0, [137].log_data[30].total := 3600.0, [137].log_data[30].time := 3600.0, [137].log_data[30].valid := 1, [137].log_data[31].max := 1.0, [137].log_data[31].total := 1440.7471, [137].log_data[31].time := 3600.0, [137].log_data[31].minminute := 1, [137].log_data[31].valid := 1, [137].log_data[32].max := 1.0, [137].log_data[32].total := 1629.7471, [137].log_data[32].time := 3600.0, [137].log_data[32].maxminute := 3, [137].log_data[32].valid := 1, [137].log_data[33].time := 3600.0, [137].log_data[33].valid := 1, [137].log_data[34].time := 3600.0, [137].log_data[34].valid := 1, [137].log_data[35].max := 1.0, [137].log_data[35].total := 1629.7471, [137].log_data[35].time := 3600.0, [137].log_data[35].maxminute := 8, [137].log_data[35].valid := 1, [137].log_data[36].max := 1.0, [137].log_data[36].total := 1527.249, [137].log_data[36].time := 3600.0, [137].log_data[36].minminute := 7, [137].log_data[36].valid := 1, [137].log_data[37].max := 7.218745, [137].log_data[37].total := 3694.3906, [137].log_data[37].time := 3600.0, [137].log_data[37].maxminute := 33, [137].log_data[37].valid := 1, [137].log_data[38].time := 3600.0, [137].log_data[38].valid := 1, [137].log_data[39].min := 0.9941174, [137].log_data[39].max := 1.0221478, [137].log_data[39].total := 3605.504, [137].log_data[39].time := 3600.0, [137].log_data[39].minminute := 11, [137].log_data[39].maxminute := 35, [137].log_data[39].valid := 1, [137].log_data[40].min := 7.5956445, [137].log_data[40].max := 7.621752, [137].log_data[40].total := 27396.43, [137].log_data[40].time := 3600.0, [137].log_data[40].minminute := 30, [137].log_data[40].maxminute := 34, [137].log_data[40].valid := 1, [137].log_data[41].min := 0.022540038, [137].log_data[41].max := 0.023128908, [137].log_data[41].total := 81.988335, [137].log_data[41].time := 3600.0, [137].log_data[41].maxminute := 40, [137].log_data[41].valid := 1, [137].log_data[42].min := 2.2911716, [137].log_data[42].max := 2.296118, [137].log_data[42].total := 8257.736, [137].log_data[42].time := 3600.0, [137].log_data[42].minminute := 43,
        [137].log_data[42].maxminute := 13, [137].log_data[42].valid := 1, [137].log_data[43].min := -0.27999878, [137].log_data[43].max := -0.26000214, [137].log_data[43].total := -953.19714, [137].log_data[43].time := 3600.0, [137].log_data[43].valid := 1, [137].log_data[44].min := -0.3199997, [137].log_data[44].max := -0.30000305, [137].log_data[44].total := -1080.1061, [137].log_data[44].time := 3600.0, [137].log_data[44].minminute := 26, [137].log_data[44].valid := 1, [137].log_data[45].time := 3600.0, [137].log_data[45].valid := 1, [137].log_data[46].time := 3600.0, [137].log_data[46].valid := 1, [137].log_data[47].time := 3600.0, [137].log_data[47].valid := 1, [137].log_data[48].min := 6.5763826, [137].log_data[48].max := 6.8665795, [137].log_data[48].total := 24016.053, [137].log_data[48].time := 3600.0, [137].log_data[48].minminute := 59, [137].log_data[48].maxminute := 38, [137].log_data[48].valid := 1, [137].log_data[49].min := 6.840525, [137].log_data[49].max := 9.479664, [137].log_data[49].total := 30308.957, [137].log_data[49].time := 3600.0, [137].log_data[49].minminute := 58, [137].log_data[49].maxminute := 35, [137].log_data[49].valid := 1, [137].log_data[50].min := 2.0497332, [137].log_data[50].max := 2.1677434, [137].log_data[50].total := 7577.8213, [137].log_data[50].time := 3600.0, [137].log_data[50].minminute := 35, [137].log_data[50].maxminute := 41, [137].log_data[50].valid := 1, [137].log_data[51].time := 3600.0, [137].log_data[51].valid := 1, [137].log_data[52].min := -2.840004, [137].log_data[52].max := 0.11999512, [137].log_data[52].total := -7516.903, [137].log_data[52].time := 3600.0, [137].log_data[52].minminute := 34, [137].log_data[52].maxminute := 1, [137].log_data[52].valid := 1, [137].log_data[53].min := -2.4600067, [137].log_data[53].max := 0.3999939, [137].log_data[53].total := -6999.097, [137].log_data[53].time := 3600.0, [137].log_data[53].minminute := 31, [137].log_data[53].maxminute := 40, [137].log_data[53].valid := 1, [137].log_data[54].max := 0.5305, [137].log_data[54].total := 1217.3619, [137].log_data[54].time := 3600.0, [137].log_data[54].minminute := 1,
        [137].log_data[54].maxminute := 34, [137].log_data[54].valid := 1, [137].log_data[55].max := 0.53, [137].log_data[55].total := 1254.2283, [137].log_data[55].time := 3600.0, [137].log_data[55].minminute := 7, [137].log_data[55].maxminute := 40, [137].log_data[55].valid := 1, [137].log_data[56].min := 0.15906787, [137].log_data[56].max := 0.1594997, [137].log_data[56].total := 573.30255, [137].log_data[56].time := 3600.0, [137].log_data[56].minminute := 5, [137].log_data[56].maxminute := 24, [137].log_data[56].valid := 1, [137].log_data[57].min := 0.20036758, [137].log_data[57].max := 0.20123126, [137].log_data[57].total := 723.45715, [137].log_data[57].time := 3600.0, [137].log_data[57].minminute := 59, [137].log_data[57].maxminute := 1, [137].log_data[57].valid := 1, [137].log_data[58].time := 3600.0, [137].log_data[58].valid := 1, [137].log_data[59].time := 3600.0, [137].log_data[59].valid := 1, [137].log_data[60].valid := 1, [137].log_data[61].valid := 1, [137].log_data[62].valid := 1, [137].log_data[63].valid := 1, [137].log_data[64].valid := 1, [137].log_data[65].valid := 1, [137].log_data[66].valid := 1, [137].log_data[67].valid := 1, [137].log_data[68].valid := 1, [137].log_data[69].valid := 1, [137].log_data[70].valid := 1, [137].log_data[71].valid := 1, [137].log_data[72].valid := 1, [137].log_data[73].valid := 1, [137].log_data[74].valid := 1, [137].log_data[75].valid := 1, [137].log_data[76].valid := 1, [137].log_data[77].valid := 1, [137].log_data[78].valid := 1, [137].log_data[79].valid := 1, [137].log_data[80].valid := 1, [137].log_data[81].valid := 1, [137].log_data[82].valid := 1, [137].log_data[83].valid := 1, [137].log_data[84].valid := 1, [137].log_data[85].valid := 1, [137].log_data[86].valid := 1, [137].log_data[87].valid := 1, [137].log_data[88].valid := 1, [137].log_data[89].valid := 1, [137].log_data[90].valid := 1, [137].log_data[91].valid := 1, [137].log_data[92].valid := 1, [137].log_data[93].valid := 1,
        [137].log_data[94].valid := 1, [137].log_data[95].valid := 1, [137].log_data[96].valid := 1, [137].log_data[97].valid := 1, [137].log_data[98].valid := 1, [137].log_data[99].valid := 1, [137].log_data[100].valid := 1, [137].log_data[101].valid := 1, [137].log_data[102].valid := 1, [137].log_data[103].valid := 1, [137].log_data[104].valid := 1, [137].log_data[105].valid := 1, [137].log_data[106].valid := 1, [137].log_data[107].valid := 1, [137].log_data[108].valid := 1, [137].log_data[109].valid := 1, [137].log_data[110].valid := 1, [137].log_data[111].valid := 1, [137].log_data[112].valid := 1, [137].log_data[113].valid := 1, [137].log_data[114].valid := 1, [137].log_data[115].valid := 1, [137].log_data[116].valid := 1, [137].log_data[117].valid := 1, [137].log_data[118].valid := 1, [137].log_data[119].valid := 1, [137].log_data[120].valid := 1, [137].log_data[121].valid := 1, [137].log_data[122].valid := 1, [137].log_data[123].valid := 1, [137].log_data[124].valid := 1, [137].time.Year := 2023, [137].time.Month := 1, [137].time.Day := 18, [137].time.Hour := 20, [137].time.Minute := 59, [137].time.Second := 59, [138].log_data[0].min := 1.0, [138].log_data[0].max := 1.0, [138].log_data[0].total := 3599.5, [138].log_data[0].time := 3599.5, [138].log_data[0].valid := 1, [138].log_data[1].max := 1.0, [138].log_data[1].total := 549.5, [138].log_data[1].time := 3599.5, [138].log_data[1].maxminute := 38, [138].log_data[1].valid := 1, [138].log_data[2].max := 1.0, [138].log_data[2].total := 546.0, [138].log_data[2].time := 3599.5, [138].log_data[2].maxminute := 38, [138].log_data[2].valid := 1, [138].log_data[3].time := 3599.5, [138].log_data[3].valid := 1, [138].log_data[4].time := 3599.5, [138].log_data[4].valid := 1, [138].log_data[5].max := 1.0, [138].log_data[5].total := 243.5, [138].log_data[5].time := 3599.5, [138].log_data[5].maxminute := 40,
        [138].log_data[5].valid := 1, [138].log_data[6].time := 3599.5, [138].log_data[6].valid := 1, [138].log_data[7].time := 3599.5, [138].log_data[7].valid := 1, [138].log_data[8].min := 1.0, [138].log_data[8].max := 1.0, [138].log_data[8].total := 3599.5, [138].log_data[8].time := 3599.5, [138].log_data[8].valid := 1, [138].log_data[9].min := 1.0, [138].log_data[9].max := 1.0, [138].log_data[9].total := 3599.5, [138].log_data[9].time := 3599.5, [138].log_data[9].valid := 1, [138].log_data[10].min := 1.0, [138].log_data[10].max := 1.0, [138].log_data[10].total := 3599.5, [138].log_data[10].time := 3599.5, [138].log_data[10].valid := 1, [138].log_data[11].time := 3599.5, [138].log_data[11].valid := 1, [138].log_data[12].min := 1.0, [138].log_data[12].max := 1.0, [138].log_data[12].total := 3599.5, [138].log_data[12].time := 3599.5, [138].log_data[12].valid := 1, [138].log_data[13].min := 1.0, [138].log_data[13].max := 1.0, [138].log_data[13].total := 3599.5, [138].log_data[13].time := 3599.5, [138].log_data[13].valid := 1, [138].log_data[14].time := 3599.5, [138].log_data[14].valid := 1, [138].log_data[15].time := 3599.5, [138].log_data[15].valid := 1, [138].log_data[16].time := 3599.5, [138].log_data[16].valid := 1, [138].log_data[17].min := 1.0, [138].log_data[17].max := 1.0, [138].log_data[17].total := 3599.5, [138].log_data[17].time := 3599.5, [138].log_data[17].valid := 1, [138].log_data[18].time := 3599.5, [138].log_data[18].valid := 1, [138].log_data[19].time := 3599.5, [138].log_data[19].valid := 1, [138].log_data[20].time := 3599.5, [138].log_data[20].valid := 1, [138].log_data[21].min := 1.0, [138].log_data[21].max := 1.0, [138].log_data[21].total := 3599.5, [138].log_data[21].time := 3599.5, [138].log_data[21].valid := 1, [138].log_data[22].time := 3599.5, [138].log_data[22].valid := 1, [138].log_data[23].time := 3599.5, [138].log_data[23].valid := 1, [138].log_data[24].time := 3599.5, [138].log_data[24].valid := 1,
        [138].log_data[25].time := 3599.5, [138].log_data[25].valid := 1, [138].log_data[26].time := 3599.5, [138].log_data[26].valid := 1, [138].log_data[27].time := 3599.5, [138].log_data[27].valid := 1, [138].log_data[28].time := 3599.5, [138].log_data[28].valid := 1, [138].log_data[29].min := 1.0, [138].log_data[29].max := 1.0, [138].log_data[29].total := 3599.5, [138].log_data[29].time := 3599.5, [138].log_data[29].valid := 1, [138].log_data[30].min := 1.0, [138].log_data[30].max := 1.0, [138].log_data[30].total := 3599.5, [138].log_data[30].time := 3599.5, [138].log_data[30].valid := 1, [138].log_data[31].max := 1.0, [138].log_data[31].total := 1439.998, [138].log_data[31].time := 3599.5, [138].log_data[31].minminute := 4, [138].log_data[31].valid := 1, [138].log_data[32].max := 1.0, [138].log_data[32].total := 1629.998, [138].log_data[32].time := 3599.5, [138].log_data[32].maxminute := 6, [138].log_data[32].valid := 1, [138].log_data[33].time := 3599.5, [138].log_data[33].valid := 1, [138].log_data[34].time := 3599.5, [138].log_data[34].valid := 1, [138].log_data[35].max := 1.0, [138].log_data[35].total := 1441.7471, [138].log_data[35].time := 3599.5, [138].log_data[35].maxminute := 11, [138].log_data[35].valid := 1, [138].log_data[36].max := 1.0, [138].log_data[36].total := 1629.7471, [138].log_data[36].time := 3599.5, [138].log_data[36].maxminute := 1, [138].log_data[36].valid := 1, [138].log_data[37].max := 7.482561, [138].log_data[37].total := 3571.9136, [138].log_data[37].time := 3599.5, [138].log_data[37].maxminute := 39, [138].log_data[37].valid := 1, [138].log_data[38].time := 3599.5, [138].log_data[38].valid := 1, [138].log_data[39].min := 0.9951773, [138].log_data[39].max := 1.02097, [138].log_data[39].total := 3605.7908, [138].log_data[39].time := 3599.5, [138].log_data[39].minminute := 55, [138].log_data[39].maxminute := 40, [138].log_data[39].valid := 1, [138].log_data[40].min := 7.6000414, [138].log_data[40].max := 7.614607, [138].log_data[40].total := 27392.58, [138].log_data[40].time := 3599.5,
        [138].log_data[40].minminute := 59, [138].log_data[40].maxminute := 54, [138].log_data[40].valid := 1, [138].log_data[41].min := 0.022540038, [138].log_data[41].max := 0.023128908, [138].log_data[41].total := 82.194374, [138].log_data[41].time := 3599.5, [138].log_data[41].maxminute := 1, [138].log_data[41].valid := 1, [138].log_data[42].min := 2.291407, [138].log_data[42].max := 2.2960005, [138].log_data[42].total := 8256.6, [138].log_data[42].time := 3599.5, [138].log_data[42].minminute := 8, [138].log_data[42].maxminute := 22, [138].log_data[42].valid := 1, [138].log_data[43].min := -0.27999878, [138].log_data[43].max := -0.26000214, [138].log_data[43].total := -961.41986, [138].log_data[43].time := 3599.5, [138].log_data[43].valid := 1, [138].log_data[44].min := -0.3199997, [138].log_data[44].max := -0.30000305, [138].log_data[44].total := -1079.9661, [138].log_data[44].time := 3599.5, [138].log_data[44].minminute := 4, [138].log_data[44].valid := 1, [138].log_data[45].time := 3599.5, [138].log_data[45].valid := 1, [138].log_data[46].time := 3599.5, [138].log_data[46].valid := 1, [138].log_data[47].time := 3599.5, [138].log_data[47].valid := 1, [138].log_data[48].min := 6.5763826, [138].log_data[48].max := 6.936381, [138].log_data[48].total := 24292.725, [138].log_data[48].time := 3599.5, [138].log_data[48].minminute := 1, [138].log_data[48].maxminute := 48, [138].log_data[48].valid := 1, [138].log_data[49].min := 6.803818, [138].log_data[49].max := 9.458463, [138].log_data[49].total := 29601.928, [138].log_data[49].time := 3599.5, [138].log_data[49].minminute := 2, [138].log_data[49].maxminute := 40, [138].log_data[49].valid := 1, [138].log_data[50].min := 2.0815325, [138].log_data[50].max := 2.2022514, [138].log_data[50].total := 7681.4053, [138].log_data[50].time := 3599.5, [138].log_data[50].minminute := 41, [138].log_data[50].maxminute := 47, [138].log_data[50].valid := 1, [138].log_data[51].time := 3599.5, [138].log_data[51].valid := 1, [138].log_data[52].min := -2.840004, [138].log_data[52].max := 0.11999512, [138].log_data[52].total := -7521.5513, [138].log_data[52].time := 3599.5,
        [138].log_data[52].minminute := 16, [138].log_data[52].maxminute := 4, [138].log_data[52].valid := 1, [138].log_data[53].min := -2.4600067, [138].log_data[53].max := 0.38000488, [138].log_data[53].total := -6813.759, [138].log_data[53].time := 3599.5, [138].log_data[53].minminute := 45, [138].log_data[53].maxminute := 42, [138].log_data[53].valid := 1, [138].log_data[54].max := 0.53, [138].log_data[54].total := 1217.2328, [138].log_data[54].time := 3599.5, [138].log_data[54].minminute := 4, [138].log_data[54].maxminute := 17, [138].log_data[54].valid := 1, [138].log_data[55].max := 0.5265, [138].log_data[55].total := 1217.1868, [138].log_data[55].time := 3599.5, [138].log_data[55].maxminute := 43, [138].log_data[55].valid := 1, [138].log_data[56].min := 0.15902862, [138].log_data[56].max := 0.1594997, [138].log_data[56].total := 573.244, [138].log_data[56].time := 3599.5, [138].log_data[56].minminute := 5, [138].log_data[56].maxminute := 10, [138].log_data[56].valid := 1, [138].log_data[57].min := 0.19860093, [138].log_data[57].max := 0.20056386, [138].log_data[57].total := 716.1004, [138].log_data[57].time := 3599.5, [138].log_data[57].minminute := 39, [138].log_data[57].valid := 1, [138].log_data[58].time := 3599.5, [138].log_data[58].valid := 1, [138].log_data[59].time := 3599.5, [138].log_data[59].valid := 1, [138].log_data[60].valid := 1, [138].log_data[61].valid := 1, [138].log_data[62].valid := 1, [138].log_data[63].valid := 1, [138].log_data[64].valid := 1, [138].log_data[65].valid := 1, [138].log_data[66].valid := 1, [138].log_data[67].valid := 1, [138].log_data[68].valid := 1, [138].log_data[69].valid := 1, [138].log_data[70].valid := 1, [138].log_data[71].valid := 1, [138].log_data[72].valid := 1, [138].log_data[73].valid := 1, [138].log_data[74].valid := 1, [138].log_data[75].valid := 1, [138].log_data[76].valid := 1, [138].log_data[77].valid := 1, [138].log_data[78].valid := 1, [138].log_data[79].valid := 1, [138].log_data[80].valid := 1, [138].log_data[81].valid := 1,
        [138].log_data[82].valid := 1, [138].log_data[83].valid := 1, [138].log_data[84].valid := 1, [138].log_data[85].valid := 1, [138].log_data[86].valid := 1, [138].log_data[87].valid := 1, [138].log_data[88].valid := 1, [138].log_data[89].valid := 1, [138].log_data[90].valid := 1, [138].log_data[91].valid := 1, [138].log_data[92].valid := 1, [138].log_data[93].valid := 1, [138].log_data[94].valid := 1, [138].log_data[95].valid := 1, [138].log_data[96].valid := 1, [138].log_data[97].valid := 1, [138].log_data[98].valid := 1, [138].log_data[99].valid := 1, [138].log_data[100].valid := 1, [138].log_data[101].valid := 1, [138].log_data[102].valid := 1, [138].log_data[103].valid := 1, [138].log_data[104].valid := 1, [138].log_data[105].valid := 1, [138].log_data[106].valid := 1, [138].log_data[107].valid := 1, [138].log_data[108].valid := 1, [138].log_data[109].valid := 1, [138].log_data[110].valid := 1, [138].log_data[111].valid := 1, [138].log_data[112].valid := 1, [138].log_data[113].valid := 1, [138].log_data[114].valid := 1, [138].log_data[115].valid := 1, [138].log_data[116].valid := 1, [138].log_data[117].valid := 1, [138].log_data[118].valid := 1, [138].log_data[119].valid := 1, [138].log_data[120].valid := 1, [138].log_data[121].valid := 1, [138].log_data[122].valid := 1, [138].log_data[123].valid := 1, [138].log_data[124].valid := 1, [138].time.Year := 2023, [138].time.Month := 1, [138].time.Day := 18, [138].time.Hour := 21, [138].time.Minute := 59, [138].time.Second := 59, [139].log_data[0].min := 1.0, [139].log_data[0].max := 1.0, [139].log_data[0].total := 3600.0, [139].log_data[0].time := 3600.0, [139].log_data[0].valid := 1, [139].log_data[1].time := 3600.0, [139].log_data[1].valid := 1, [139].log_data[2].time := 3600.0, [139].log_data[2].valid := 1, [139].log_data[3].time := 3600.0, [139].log_data[3].valid := 1,
        [139].log_data[4].time := 3600.0, [139].log_data[4].valid := 1, [139].log_data[5].time := 3600.0, [139].log_data[5].valid := 1, [139].log_data[6].time := 3600.0, [139].log_data[6].valid := 1, [139].log_data[7].time := 3600.0, [139].log_data[7].valid := 1, [139].log_data[8].min := 1.0, [139].log_data[8].max := 1.0, [139].log_data[8].total := 3600.0, [139].log_data[8].time := 3600.0, [139].log_data[8].valid := 1, [139].log_data[9].min := 1.0, [139].log_data[9].max := 1.0, [139].log_data[9].total := 3600.0, [139].log_data[9].time := 3600.0, [139].log_data[9].valid := 1, [139].log_data[10].min := 1.0, [139].log_data[10].max := 1.0, [139].log_data[10].total := 3600.0, [139].log_data[10].time := 3600.0, [139].log_data[10].valid := 1, [139].log_data[11].time := 3600.0, [139].log_data[11].valid := 1, [139].log_data[12].min := 1.0, [139].log_data[12].max := 1.0, [139].log_data[12].total := 3600.0, [139].log_data[12].time := 3600.0, [139].log_data[12].valid := 1, [139].log_data[13].min := 1.0, [139].log_data[13].max := 1.0, [139].log_data[13].total := 3600.0, [139].log_data[13].time := 3600.0, [139].log_data[13].valid := 1, [139].log_data[14].time := 3600.0, [139].log_data[14].valid := 1, [139].log_data[15].time := 3600.0, [139].log_data[15].valid := 1, [139].log_data[16].time := 3600.0, [139].log_data[16].valid := 1, [139].log_data[17].min := 1.0, [139].log_data[17].max := 1.0, [139].log_data[17].total := 3600.0, [139].log_data[17].time := 3600.0, [139].log_data[17].valid := 1, [139].log_data[18].time := 3600.0, [139].log_data[18].valid := 1, [139].log_data[19].time := 3600.0, [139].log_data[19].valid := 1, [139].log_data[20].time := 3600.0, [139].log_data[20].valid := 1, [139].log_data[21].min := 1.0, [139].log_data[21].max := 1.0, [139].log_data[21].total := 3600.0, [139].log_data[21].time := 3600.0, [139].log_data[21].valid := 1, [139].log_data[22].time := 3600.0, [139].log_data[22].valid := 1, [139].log_data[23].time := 3600.0,
        [139].log_data[23].valid := 1, [139].log_data[24].time := 3600.0, [139].log_data[24].valid := 1, [139].log_data[25].time := 3600.0, [139].log_data[25].valid := 1, [139].log_data[26].time := 3600.0, [139].log_data[26].valid := 1, [139].log_data[27].time := 3600.0, [139].log_data[27].valid := 1, [139].log_data[28].time := 3600.0, [139].log_data[28].valid := 1, [139].log_data[29].min := 1.0, [139].log_data[29].max := 1.0, [139].log_data[29].total := 3600.0, [139].log_data[29].time := 3600.0, [139].log_data[29].valid := 1, [139].log_data[30].min := 1.0, [139].log_data[30].max := 1.0, [139].log_data[30].total := 3600.0, [139].log_data[30].time := 3600.0, [139].log_data[30].valid := 1, [139].log_data[31].max := 1.0, [139].log_data[31].total := 1569.998, [139].log_data[31].time := 3600.0, [139].log_data[31].minminute := 8, [139].log_data[31].valid := 1, [139].log_data[32].max := 1.0, [139].log_data[32].total := 1588.998, [139].log_data[32].time := 3600.0, [139].log_data[32].maxminute := 9, [139].log_data[32].valid := 1, [139].log_data[33].time := 3600.0, [139].log_data[33].valid := 1, [139].log_data[34].time := 3600.0, [139].log_data[34].valid := 1, [139].log_data[35].max := 1.0, [139].log_data[35].total := 1440.7471, [139].log_data[35].time := 3600.0, [139].log_data[35].minminute := 3, [139].log_data[35].valid := 1, [139].log_data[36].max := 1.0, [139].log_data[36].total := 1629.7471, [139].log_data[36].time := 3600.0, [139].log_data[36].maxminute := 4, [139].log_data[36].valid := 1, [139].log_data[37].time := 3600.0, [139].log_data[37].valid := 1, [139].log_data[38].time := 3600.0, [139].log_data[38].valid := 1, [139].log_data[39].min := 0.9936463, [139].log_data[39].max := 1.0022438, [139].log_data[39].total := 3595.2498, [139].log_data[39].time := 3600.0, [139].log_data[39].minminute := 9, [139].log_data[39].maxminute := 48, [139].log_data[39].valid := 1, [139].log_data[40].min := 7.585752, [139].log_data[40].max := 7.630545, [139].log_data[40].total := 27394.008, [139].log_data[40].time := 3600.0,
        [139].log_data[40].minminute := 7, [139].log_data[40].maxminute := 12, [139].log_data[40].valid := 1, [139].log_data[41].min := 0.022540038, [139].log_data[41].max := 0.023128908, [139].log_data[41].total := 82.32532, [139].log_data[41].time := 3600.0, [139].log_data[41].minminute := 4, [139].log_data[41].maxminute := 20, [139].log_data[41].valid := 1, [139].log_data[42].min := 2.290936, [139].log_data[42].max := 2.2958827, [139].log_data[42].total := 8257.735, [139].log_data[42].time := 3600.0, [139].log_data[42].minminute := 45, [139].log_data[42].maxminute := 30, [139].log_data[42].valid := 1, [139].log_data[43].min := -0.27999878, [139].log_data[43].max := -0.26000214, [139].log_data[43].total := -953.62024, [139].log_data[43].time := 3600.0, [139].log_data[43].valid := 1, [139].log_data[44].min := -0.30000305, [139].log_data[44].max := -0.27999878, [139].log_data[44].total := -1080.086, [139].log_data[44].time := 3600.0, [139].log_data[44].maxminute := 42, [139].log_data[44].valid := 1, [139].log_data[45].time := 3600.0, [139].log_data[45].valid := 1, [139].log_data[46].time := 3600.0, [139].log_data[46].valid := 1, [139].log_data[47].time := 3600.0, [139].log_data[47].valid := 1, [139].log_data[48].min := 6.58655, [139].log_data[48].max := 6.792656, [139].log_data[48].total := 24205.99, [139].log_data[48].time := 3600.0, [139].log_data[48].minminute := 12, [139].log_data[48].maxminute := 25, [139].log_data[48].valid := 1, [139].log_data[49].min := 6.8130445, [139].log_data[49].max := 9.584482, [139].log_data[49].total := 30477.682, [139].log_data[49].time := 3600.0, [139].log_data[49].minminute := 9, [139].log_data[49].maxminute := 58, [139].log_data[49].valid := 1, [139].log_data[50].min := 2.0974321, [139].log_data[50].max := 2.186941, [139].log_data[50].total := 7713.532, [139].log_data[50].time := 3600.0, [139].log_data[50].minminute := 58, [139].log_data[50].valid := 1, [139].log_data[51].time := 3600.0, [139].log_data[51].valid := 1, [139].log_data[52].min := -2.7799988, [139].log_data[52].max := 0.11999512, [139].log_data[52].total := -7817.1143, [139].log_data[52].time := 3600.0,
        [139].log_data[52].minminute := 41, [139].log_data[52].maxminute := 8, [139].log_data[52].valid := 1, [139].log_data[53].min := -2.4400024, [139].log_data[53].max := 0.3999939, [139].log_data[53].total := -6833.1123, [139].log_data[53].time := 3600.0, [139].log_data[53].minminute := 27, [139].log_data[53].maxminute := 46, [139].log_data[53].valid := 1, [139].log_data[54].max := 0.5255, [139].log_data[54].total := 1254.3971, [139].log_data[54].time := 3600.0, [139].log_data[54].minminute := 8, [139].log_data[54].maxminute := 41, [139].log_data[54].valid := 1, [139].log_data[55].max := 0.5435, [139].log_data[55].total := 1217.3762, [139].log_data[55].time := 3600.0, [139].log_data[55].minminute := 3, [139].log_data[55].maxminute := 57, [139].log_data[55].valid := 1, [139].log_data[56].min := 0.15910713, [139].log_data[56].max := 0.15953897, [139].log_data[56].total := 573.45483, [139].log_data[56].time := 3600.0, [139].log_data[56].minminute := 13, [139].log_data[56].maxminute := 27, [139].log_data[56].valid := 1, [139].log_data[57].min := 0.19671655, [139].log_data[57].max := 0.19899355, [139].log_data[57].total := 710.38025, [139].log_data[57].time := 3600.0, [139].log_data[57].minminute := 25, [139].log_data[57].valid := 1, [139].log_data[58].time := 3600.0, [139].log_data[58].valid := 1, [139].log_data[59].time := 3600.0, [139].log_data[59].valid := 1, [139].log_data[60].valid := 1, [139].log_data[61].valid := 1, [139].log_data[62].valid := 1, [139].log_data[63].valid := 1, [139].log_data[64].valid := 1, [139].log_data[65].valid := 1, [139].log_data[66].valid := 1, [139].log_data[67].valid := 1, [139].log_data[68].valid := 1, [139].log_data[69].valid := 1, [139].log_data[70].valid := 1, [139].log_data[71].valid := 1, [139].log_data[72].valid := 1, [139].log_data[73].valid := 1, [139].log_data[74].valid := 1, [139].log_data[75].valid := 1, [139].log_data[76].valid := 1, [139].log_data[77].valid := 1, [139].log_data[78].valid := 1, [139].log_data[79].valid := 1, [139].log_data[80].valid := 1,
        [139].log_data[81].valid := 1, [139].log_data[82].valid := 1, [139].log_data[83].valid := 1, [139].log_data[84].valid := 1, [139].log_data[85].valid := 1, [139].log_data[86].valid := 1, [139].log_data[87].valid := 1, [139].log_data[88].valid := 1, [139].log_data[89].valid := 1, [139].log_data[90].valid := 1, [139].log_data[91].valid := 1, [139].log_data[92].valid := 1, [139].log_data[93].valid := 1, [139].log_data[94].valid := 1, [139].log_data[95].valid := 1, [139].log_data[96].valid := 1, [139].log_data[97].valid := 1, [139].log_data[98].valid := 1, [139].log_data[99].valid := 1, [139].log_data[100].valid := 1, [139].log_data[101].valid := 1, [139].log_data[102].valid := 1, [139].log_data[103].valid := 1, [139].log_data[104].valid := 1, [139].log_data[105].valid := 1, [139].log_data[106].valid := 1, [139].log_data[107].valid := 1, [139].log_data[108].valid := 1, [139].log_data[109].valid := 1, [139].log_data[110].valid := 1, [139].log_data[111].valid := 1, [139].log_data[112].valid := 1, [139].log_data[113].valid := 1, [139].log_data[114].valid := 1, [139].log_data[115].valid := 1, [139].log_data[116].valid := 1, [139].log_data[117].valid := 1, [139].log_data[118].valid := 1, [139].log_data[119].valid := 1, [139].log_data[120].valid := 1, [139].log_data[121].valid := 1, [139].log_data[122].valid := 1, [139].log_data[123].valid := 1, [139].log_data[124].valid := 1, [139].time.Year := 2023, [139].time.Month := 1, [139].time.Day := 18, [139].time.Hour := 22, [139].time.Minute := 59, [139].time.Second := 59, [140].log_data[0].min := 1.0, [140].log_data[0].max := 1.0, [140].log_data[0].total := 3600.0, [140].log_data[0].time := 3600.0, [140].log_data[0].valid := 1, [140].log_data[1].max := 1.0, [140].log_data[1].total := 561.0, [140].log_data[1].time := 3600.0, [140].log_data[1].maxminute := 17, [140].log_data[1].valid := 1,
        [140].log_data[2].max := 1.0, [140].log_data[2].total := 557.5, [140].log_data[2].time := 3600.0, [140].log_data[2].maxminute := 17, [140].log_data[2].valid := 1, [140].log_data[3].time := 3600.0, [140].log_data[3].valid := 1, [140].log_data[4].time := 3600.0, [140].log_data[4].valid := 1, [140].log_data[5].max := 1.0, [140].log_data[5].total := 235.5, [140].log_data[5].time := 3600.0, [140].log_data[5].maxminute := 20, [140].log_data[5].valid := 1, [140].log_data[6].time := 3600.0, [140].log_data[6].valid := 1, [140].log_data[7].time := 3600.0, [140].log_data[7].valid := 1, [140].log_data[8].min := 1.0, [140].log_data[8].max := 1.0, [140].log_data[8].total := 3600.0, [140].log_data[8].time := 3600.0, [140].log_data[8].valid := 1, [140].log_data[9].min := 1.0, [140].log_data[9].max := 1.0, [140].log_data[9].total := 3600.0, [140].log_data[9].time := 3600.0, [140].log_data[9].valid := 1, [140].log_data[10].min := 1.0, [140].log_data[10].max := 1.0, [140].log_data[10].total := 3600.0, [140].log_data[10].time := 3600.0, [140].log_data[10].valid := 1, [140].log_data[11].time := 3600.0, [140].log_data[11].valid := 1, [140].log_data[12].min := 1.0, [140].log_data[12].max := 1.0, [140].log_data[12].total := 3600.0, [140].log_data[12].time := 3600.0, [140].log_data[12].valid := 1, [140].log_data[13].min := 1.0, [140].log_data[13].max := 1.0, [140].log_data[13].total := 3600.0, [140].log_data[13].time := 3600.0, [140].log_data[13].valid := 1, [140].log_data[14].time := 3600.0, [140].log_data[14].valid := 1, [140].log_data[15].time := 3600.0, [140].log_data[15].valid := 1, [140].log_data[16].time := 3600.0, [140].log_data[16].valid := 1, [140].log_data[17].min := 1.0, [140].log_data[17].max := 1.0, [140].log_data[17].total := 3600.0, [140].log_data[17].time := 3600.0, [140].log_data[17].valid := 1, [140].log_data[18].time := 3600.0, [140].log_data[18].valid := 1, [140].log_data[19].time := 3600.0, [140].log_data[19].valid := 1,
        [140].log_data[20].time := 3600.0, [140].log_data[20].valid := 1, [140].log_data[21].min := 1.0, [140].log_data[21].max := 1.0, [140].log_data[21].total := 3600.0, [140].log_data[21].time := 3600.0, [140].log_data[21].valid := 1, [140].log_data[22].time := 3600.0, [140].log_data[22].valid := 1, [140].log_data[23].time := 3600.0, [140].log_data[23].valid := 1, [140].log_data[24].time := 3600.0, [140].log_data[24].valid := 1, [140].log_data[25].time := 3600.0, [140].log_data[25].valid := 1, [140].log_data[26].time := 3600.0, [140].log_data[26].valid := 1, [140].log_data[27].time := 3600.0, [140].log_data[27].valid := 1, [140].log_data[28].time := 3600.0, [140].log_data[28].valid := 1, [140].log_data[29].min := 1.0, [140].log_data[29].max := 1.0, [140].log_data[29].total := 3600.0, [140].log_data[29].time := 3600.0, [140].log_data[29].valid := 1, [140].log_data[30].min := 1.0, [140].log_data[30].max := 1.0, [140].log_data[30].total := 3600.0, [140].log_data[30].time := 3600.0, [140].log_data[30].valid := 1, [140].log_data[31].max := 1.0, [140].log_data[31].total := 1629.7471, [140].log_data[31].time := 3600.0, [140].log_data[31].maxminute := 2, [140].log_data[31].valid := 1, [140].log_data[32].max := 1.0, [140].log_data[32].total := 1440.998, [140].log_data[32].time := 3600.0, [140].log_data[32].valid := 1, [140].log_data[33].time := 3600.0, [140].log_data[33].valid := 1, [140].log_data[34].time := 3600.0, [140].log_data[34].valid := 1, [140].log_data[35].max := 1.0, [140].log_data[35].total := 1463.498, [140].log_data[35].time := 3600.0, [140].log_data[35].minminute := 6, [140].log_data[35].valid := 1, [140].log_data[36].max := 1.0, [140].log_data[36].total := 1629.7471, [140].log_data[36].time := 3600.0, [140].log_data[36].maxminute := 7, [140].log_data[36].valid := 1, [140].log_data[37].max := 7.2297378, [140].log_data[37].total := 3526.3813, [140].log_data[37].time := 3600.0, [140].log_data[37].maxminute := 19, [140].log_data[37].valid := 1, [140].log_data[38].time := 3600.0,
        [140].log_data[38].valid := 1, [140].log_data[39].min := 0.9945885, [140].log_data[39].max := 1.0215589, [140].log_data[39].total := 3602.9668, [140].log_data[39].time := 3600.0, [140].log_data[39].minminute := 57, [140].log_data[39].maxminute := 25, [140].log_data[39].valid := 1, [140].log_data[40].min := 7.6041636, [140].log_data[40].max := 7.617629, [140].log_data[40].total := 27402.25, [140].log_data[40].time := 3600.0, [140].log_data[40].minminute := 34, [140].log_data[40].maxminute := 6, [140].log_data[40].valid := 1, [140].log_data[41].min := 0.02273633, [140].log_data[41].max := 0.023128908, [140].log_data[41].total := 82.444305, [140].log_data[41].time := 3600.0, [140].log_data[41].valid := 1, [140].log_data[42].min := 2.291525, [140].log_data[42].max := 2.2958827, [140].log_data[42].total := 8257.811, [140].log_data[42].time := 3600.0, [140].log_data[42].minminute := 14, [140].log_data[42].maxminute := 12, [140].log_data[42].valid := 1, [140].log_data[43].min := -0.27999878, [140].log_data[43].max := -0.26000214, [140].log_data[43].total := -957.4939, [140].log_data[43].time := 3600.0, [140].log_data[43].valid := 1, [140].log_data[44].min := -0.3199997, [140].log_data[44].max := -0.30000305, [140].log_data[44].total := -1080.1212, [140].log_data[44].time := 3600.0, [140].log_data[44].minminute := 23, [140].log_data[44].valid := 1, [140].log_data[45].time := 3600.0, [140].log_data[45].valid := 1, [140].log_data[46].time := 3600.0, [140].log_data[46].valid := 1, [140].log_data[47].time := 3600.0, [140].log_data[47].valid := 1, [140].log_data[48].min := 6.590947, [140].log_data[48].max := 6.9591894, [140].log_data[48].total := 24227.748, [140].log_data[48].time := 3600.0, [140].log_data[48].minminute := 51, [140].log_data[48].maxminute := 27, [140].log_data[48].valid := 1, [140].log_data[49].min := 6.937297, [140].log_data[49].max := 9.630414, [140].log_data[49].total := 30100.4, [140].log_data[49].time := 3600.0, [140].log_data[49].minminute := 49, [140].log_data[49].maxminute := 16, [140].log_data[49].valid := 1, [140].log_data[50].min := 2.0675173, [140].log_data[50].max := 2.1808167,
        [140].log_data[50].total := 7664.448, [140].log_data[50].time := 3600.0, [140].log_data[50].minminute := 20, [140].log_data[50].maxminute := 27, [140].log_data[50].valid := 1, [140].log_data[51].time := 3600.0, [140].log_data[51].valid := 1, [140].log_data[52].min := -2.8199997, [140].log_data[52].max := 0.11999512, [140].log_data[52].total := -7578.174, [140].log_data[52].time := 3600.0, [140].log_data[52].minminute := 44, [140].log_data[52].valid := 1, [140].log_data[53].min := -2.4600067, [140].log_data[53].max := 0.3600006, [140].log_data[53].total := -6987.451, [140].log_data[53].time := 3600.0, [140].log_data[53].minminute := 3, [140].log_data[53].maxminute := 7, [140].log_data[53].valid := 1, [140].log_data[54].max := 0.5305, [140].log_data[54].total := 1217.1968, [140].log_data[54].time := 3600.0, [140].log_data[54].maxminute := 44, [140].log_data[54].valid := 1, [140].log_data[55].max := 0.524, [140].log_data[55].total := 1228.1274, [140].log_data[55].time := 3600.0, [140].log_data[55].minminute := 6, [140].log_data[55].maxminute := 18, [140].log_data[55].valid := 1, [140].log_data[56].min := 0.15910713, [140].log_data[56].max := 0.15957822, [140].log_data[56].total := 573.4776, [140].log_data[56].time := 3600.0, [140].log_data[56].minminute := 57, [140].log_data[56].maxminute := 14, [140].log_data[56].valid := 1, [140].log_data[57].min := 0.19510698, [140].log_data[57].max := 0.19710913, [140].log_data[57].total := 708.2146, [140].log_data[57].time := 3600.0, [140].log_data[57].minminute := 59, [140].log_data[57].maxminute := 2, [140].log_data[57].valid := 1, [140].log_data[58].time := 3600.0, [140].log_data[58].valid := 1, [140].log_data[59].time := 3600.0, [140].log_data[59].valid := 1, [140].log_data[60].valid := 1, [140].log_data[61].valid := 1, [140].log_data[62].valid := 1, [140].log_data[63].valid := 1, [140].log_data[64].valid := 1, [140].log_data[65].valid := 1, [140].log_data[66].valid := 1, [140].log_data[67].valid := 1, [140].log_data[68].valid := 1, [140].log_data[69].valid := 1, [140].log_data[70].valid := 1,
        [140].log_data[71].valid := 1, [140].log_data[72].valid := 1, [140].log_data[73].valid := 1, [140].log_data[74].valid := 1, [140].log_data[75].valid := 1, [140].log_data[76].valid := 1, [140].log_data[77].valid := 1, [140].log_data[78].valid := 1, [140].log_data[79].valid := 1, [140].log_data[80].valid := 1, [140].log_data[81].valid := 1, [140].log_data[82].valid := 1, [140].log_data[83].valid := 1, [140].log_data[84].valid := 1, [140].log_data[85].valid := 1, [140].log_data[86].valid := 1, [140].log_data[87].valid := 1, [140].log_data[88].valid := 1, [140].log_data[89].valid := 1, [140].log_data[90].valid := 1, [140].log_data[91].valid := 1, [140].log_data[92].valid := 1, [140].log_data[93].valid := 1, [140].log_data[94].valid := 1, [140].log_data[95].valid := 1, [140].log_data[96].valid := 1, [140].log_data[97].valid := 1, [140].log_data[98].valid := 1, [140].log_data[99].valid := 1, [140].log_data[100].valid := 1, [140].log_data[101].valid := 1, [140].log_data[102].valid := 1, [140].log_data[103].valid := 1, [140].log_data[104].valid := 1, [140].log_data[105].valid := 1, [140].log_data[106].valid := 1, [140].log_data[107].valid := 1, [140].log_data[108].valid := 1, [140].log_data[109].valid := 1, [140].log_data[110].valid := 1, [140].log_data[111].valid := 1, [140].log_data[112].valid := 1, [140].log_data[113].valid := 1, [140].log_data[114].valid := 1, [140].log_data[115].valid := 1, [140].log_data[116].valid := 1, [140].log_data[117].valid := 1, [140].log_data[118].valid := 1, [140].log_data[119].valid := 1, [140].log_data[120].valid := 1, [140].log_data[121].valid := 1, [140].log_data[122].valid := 1, [140].log_data[123].valid := 1, [140].log_data[124].valid := 1, [140].time.Year := 2023, [140].time.Month := 1, [140].time.Day := 18, [140].time.Hour := 23, [140].time.Minute := 59, [140].time.Second := 59,
        [141].log_data[0].min := 1.0, [141].log_data[0].max := 1.0, [141].log_data[0].total := 3600.0, [141].log_data[0].time := 3600.0, [141].log_data[0].valid := 1, [141].log_data[1].time := 3600.0, [141].log_data[1].valid := 1, [141].log_data[2].time := 3600.0, [141].log_data[2].valid := 1, [141].log_data[3].time := 3600.0, [141].log_data[3].valid := 1, [141].log_data[4].time := 3600.0, [141].log_data[4].valid := 1, [141].log_data[5].time := 3600.0, [141].log_data[5].valid := 1, [141].log_data[6].time := 3600.0, [141].log_data[6].valid := 1, [141].log_data[7].time := 3600.0, [141].log_data[7].valid := 1, [141].log_data[8].min := 1.0, [141].log_data[8].max := 1.0, [141].log_data[8].total := 3600.0, [141].log_data[8].time := 3600.0, [141].log_data[8].valid := 1, [141].log_data[9].min := 1.0, [141].log_data[9].max := 1.0, [141].log_data[9].total := 3600.0, [141].log_data[9].time := 3600.0, [141].log_data[9].valid := 1, [141].log_data[10].min := 1.0, [141].log_data[10].max := 1.0, [141].log_data[10].total := 3600.0, [141].log_data[10].time := 3600.0, [141].log_data[10].valid := 1, [141].log_data[11].time := 3600.0, [141].log_data[11].valid := 1, [141].log_data[12].min := 1.0, [141].log_data[12].max := 1.0, [141].log_data[12].total := 3600.0, [141].log_data[12].time := 3600.0, [141].log_data[12].valid := 1, [141].log_data[13].min := 1.0, [141].log_data[13].max := 1.0, [141].log_data[13].total := 3600.0, [141].log_data[13].time := 3600.0, [141].log_data[13].valid := 1, [141].log_data[14].time := 3600.0, [141].log_data[14].valid := 1, [141].log_data[15].time := 3600.0, [141].log_data[15].valid := 1, [141].log_data[16].time := 3600.0, [141].log_data[16].valid := 1, [141].log_data[17].min := 1.0, [141].log_data[17].max := 1.0, [141].log_data[17].total := 3600.0, [141].log_data[17].time := 3600.0, [141].log_data[17].valid := 1, [141].log_data[18].time := 3600.0, [141].log_data[18].valid := 1, [141].log_data[19].time := 3600.0,
        [141].log_data[19].valid := 1, [141].log_data[20].time := 3600.0, [141].log_data[20].valid := 1, [141].log_data[21].min := 1.0, [141].log_data[21].max := 1.0, [141].log_data[21].total := 3600.0, [141].log_data[21].time := 3600.0, [141].log_data[21].valid := 1, [141].log_data[22].time := 3600.0, [141].log_data[22].valid := 1, [141].log_data[23].time := 3600.0, [141].log_data[23].valid := 1, [141].log_data[24].time := 3600.0, [141].log_data[24].valid := 1, [141].log_data[25].time := 3600.0, [141].log_data[25].valid := 1, [141].log_data[26].time := 3600.0, [141].log_data[26].valid := 1, [141].log_data[27].time := 3600.0, [141].log_data[27].valid := 1, [141].log_data[28].time := 3600.0, [141].log_data[28].valid := 1, [141].log_data[29].min := 1.0, [141].log_data[29].max := 1.0, [141].log_data[29].total := 3600.0, [141].log_data[29].time := 3600.0, [141].log_data[29].valid := 1, [141].log_data[30].min := 1.0, [141].log_data[30].max := 1.0, [141].log_data[30].total := 3600.0, [141].log_data[30].time := 3600.0, [141].log_data[30].valid := 1, [141].log_data[31].max := 1.0, [141].log_data[31].total := 1629.998, [141].log_data[31].time := 3600.0, [141].log_data[31].maxminute := 5, [141].log_data[31].valid := 1, [141].log_data[32].max := 1.0, [141].log_data[32].total := 1440.7471, [141].log_data[32].time := 3600.0, [141].log_data[32].minminute := 3, [141].log_data[32].valid := 1, [141].log_data[33].time := 3600.0, [141].log_data[33].valid := 1, [141].log_data[34].time := 3600.0, [141].log_data[34].valid := 1, [141].log_data[35].max := 1.0, [141].log_data[35].total := 1629.7471, [141].log_data[35].time := 3600.0, [141].log_data[35].valid := 1, [141].log_data[36].max := 1.0, [141].log_data[36].total := 1506.2471, [141].log_data[36].time := 3600.0, [141].log_data[36].maxminute := 10, [141].log_data[36].valid := 1, [141].log_data[37].time := 3600.0, [141].log_data[37].valid := 1, [141].log_data[38].time := 3600.0, [141].log_data[38].valid := 1, [141].log_data[39].min := 0.9945885,
        [141].log_data[39].max := 1.0034214, [141].log_data[39].total := 3598.7166, [141].log_data[39].time := 3600.0, [141].log_data[39].minminute := 14, [141].log_data[39].maxminute := 23, [141].log_data[39].valid := 1, [141].log_data[40].min := 7.602789, [141].log_data[40].max := 7.6165304, [141].log_data[40].total := 27404.78, [141].log_data[40].time := 3600.0, [141].log_data[40].minminute := 22, [141].log_data[40].maxminute := 26, [141].log_data[40].valid := 1, [141].log_data[41].min := 0.02273633, [141].log_data[41].max := 0.023128908, [141].log_data[41].total := 82.49746, [141].log_data[41].time := 3600.0, [141].log_data[41].valid := 1, [141].log_data[42].min := 2.291407, [141].log_data[42].max := 2.2958827, [141].log_data[42].total := 8257.892, [141].log_data[42].time := 3600.0, [141].log_data[42].minminute := 36, [141].log_data[42].valid := 1, [141].log_data[43].min := -0.27999878, [141].log_data[43].max := -0.26000214, [141].log_data[43].total := -1000.8294, [141].log_data[43].time := 3600.0, [141].log_data[43].valid := 1, [141].log_data[44].min := -0.3199997, [141].log_data[44].max := -0.30000305, [141].log_data[44].total := -1082.3021, [141].log_data[44].time := 3600.0, [141].log_data[44].minminute := 6, [141].log_data[44].valid := 1, [141].log_data[45].time := 3600.0, [141].log_data[45].valid := 1, [141].log_data[46].time := 3600.0, [141].log_data[46].valid := 1, [141].log_data[47].time := 3600.0, [141].log_data[47].valid := 1, [141].log_data[48].min := 6.703893, [141].log_data[48].max := 6.808595, [141].log_data[48].total := 24397.516, [141].log_data[48].time := 3600.0, [141].log_data[48].maxminute := 6, [141].log_data[48].valid := 1, [141].log_data[49].min := 8.0222, [141].log_data[49].max := 9.619422, [141].log_data[49].total := 33614.934, [141].log_data[49].time := 3600.0, [141].log_data[49].maxminute := 57, [141].log_data[49].valid := 1, [141].log_data[50].min := 2.0484376, [141].log_data[50].max := 2.1406553, [141].log_data[50].total := 7540.1885, [141].log_data[50].time := 3600.0, [141].log_data[50].minminute := 58, [141].log_data[50].valid := 1, [141].log_data[51].time := 3600.0,
        [141].log_data[51].valid := 1, [141].log_data[52].min := -2.880005, [141].log_data[52].max := 0.11999512, [141].log_data[52].total := -7609.968, [141].log_data[52].time := 3600.0, [141].log_data[52].minminute := 36, [141].log_data[52].maxminute := 3, [141].log_data[52].valid := 1, [141].log_data[53].min := -2.4800034, [141].log_data[53].max := 0.38000488, [141].log_data[53].total := -7040.133, [141].log_data[53].time := 3600.0, [141].log_data[53].maxminute := 52, [141].log_data[53].valid := 1, [141].log_data[54].max := 0.538, [141].log_data[54].total := 1217.3525, [141].log_data[54].time := 3600.0, [141].log_data[54].minminute := 3, [141].log_data[54].maxminute := 36, [141].log_data[54].valid := 1, [141].log_data[55].max := 0.538, [141].log_data[55].total := 1243.2715, [141].log_data[55].time := 3600.0, [141].log_data[55].valid := 1, [141].log_data[56].min := 0.15906787, [141].log_data[56].max := 0.15961748, [141].log_data[56].total := 573.5186, [141].log_data[56].time := 3600.0, [141].log_data[56].minminute := 30, [141].log_data[56].maxminute := 23, [141].log_data[56].valid := 1, [141].log_data[57].min := 0.19494995, [141].log_data[57].max := 0.19542104, [141].log_data[57].total := 702.5909, [141].log_data[57].time := 3600.0, [141].log_data[57].minminute := 55, [141].log_data[57].maxminute := 15, [141].log_data[57].valid := 1, [141].log_data[58].time := 3600.0, [141].log_data[58].valid := 1, [141].log_data[59].time := 3600.0, [141].log_data[59].valid := 1, [141].log_data[60].valid := 1, [141].log_data[61].valid := 1, [141].log_data[62].valid := 1, [141].log_data[63].valid := 1, [141].log_data[64].valid := 1, [141].log_data[65].valid := 1, [141].log_data[66].valid := 1, [141].log_data[67].valid := 1, [141].log_data[68].valid := 1, [141].log_data[69].valid := 1, [141].log_data[70].valid := 1, [141].log_data[71].valid := 1, [141].log_data[72].valid := 1, [141].log_data[73].valid := 1, [141].log_data[74].valid := 1, [141].log_data[75].valid := 1, [141].log_data[76].valid := 1, [141].log_data[77].valid := 1,
        [141].log_data[78].valid := 1, [141].log_data[79].valid := 1, [141].log_data[80].valid := 1, [141].log_data[81].valid := 1, [141].log_data[82].valid := 1, [141].log_data[83].valid := 1, [141].log_data[84].valid := 1, [141].log_data[85].valid := 1, [141].log_data[86].valid := 1, [141].log_data[87].valid := 1, [141].log_data[88].valid := 1, [141].log_data[89].valid := 1, [141].log_data[90].valid := 1, [141].log_data[91].valid := 1, [141].log_data[92].valid := 1, [141].log_data[93].valid := 1, [141].log_data[94].valid := 1, [141].log_data[95].valid := 1, [141].log_data[96].valid := 1, [141].log_data[97].valid := 1, [141].log_data[98].valid := 1, [141].log_data[99].valid := 1, [141].log_data[100].valid := 1, [141].log_data[101].valid := 1, [141].log_data[102].valid := 1, [141].log_data[103].valid := 1, [141].log_data[104].valid := 1, [141].log_data[105].valid := 1, [141].log_data[106].valid := 1, [141].log_data[107].valid := 1, [141].log_data[108].valid := 1, [141].log_data[109].valid := 1, [141].log_data[110].valid := 1, [141].log_data[111].valid := 1, [141].log_data[112].valid := 1, [141].log_data[113].valid := 1, [141].log_data[114].valid := 1, [141].log_data[115].valid := 1, [141].log_data[116].valid := 1, [141].log_data[117].valid := 1, [141].log_data[118].valid := 1, [141].log_data[119].valid := 1, [141].log_data[120].valid := 1, [141].log_data[121].valid := 1, [141].log_data[122].valid := 1, [141].log_data[123].valid := 1, [141].log_data[124].valid := 1, [141].time.Year := 2023, [141].time.Month := 1, [141].time.Day := 19, [141].time.Minute := 59, [141].time.Second := 59, [142].log_data[0].min := 1.0, [142].log_data[0].max := 1.0, [142].log_data[0].total := 3600.0, [142].log_data[0].time := 3600.0, [142].log_data[0].valid := 1, [142].log_data[1].max := 1.0, [142].log_data[1].total := 532.5, [142].log_data[1].time := 3600.0,
        [142].log_data[1].maxminute := 13, [142].log_data[1].valid := 1, [142].log_data[2].max := 1.0, [142].log_data[2].total := 529.0, [142].log_data[2].time := 3600.0, [142].log_data[2].maxminute := 13, [142].log_data[2].valid := 1, [142].log_data[3].time := 3600.0, [142].log_data[3].valid := 1, [142].log_data[4].time := 3600.0, [142].log_data[4].valid := 1, [142].log_data[5].max := 1.0, [142].log_data[5].total := 228.0, [142].log_data[5].time := 3600.0, [142].log_data[5].maxminute := 15, [142].log_data[5].valid := 1, [142].log_data[6].time := 3600.0, [142].log_data[6].valid := 1, [142].log_data[7].time := 3600.0, [142].log_data[7].valid := 1, [142].log_data[8].min := 1.0, [142].log_data[8].max := 1.0, [142].log_data[8].total := 3600.0, [142].log_data[8].time := 3600.0, [142].log_data[8].valid := 1, [142].log_data[9].min := 1.0, [142].log_data[9].max := 1.0, [142].log_data[9].total := 3600.0, [142].log_data[9].time := 3600.0, [142].log_data[9].valid := 1, [142].log_data[10].min := 1.0, [142].log_data[10].max := 1.0, [142].log_data[10].total := 3600.0, [142].log_data[10].time := 3600.0, [142].log_data[10].valid := 1, [142].log_data[11].time := 3600.0, [142].log_data[11].valid := 1, [142].log_data[12].min := 1.0, [142].log_data[12].max := 1.0, [142].log_data[12].total := 3600.0, [142].log_data[12].time := 3600.0, [142].log_data[12].valid := 1, [142].log_data[13].min := 1.0, [142].log_data[13].max := 1.0, [142].log_data[13].total := 3600.0, [142].log_data[13].time := 3600.0, [142].log_data[13].valid := 1, [142].log_data[14].time := 3600.0, [142].log_data[14].valid := 1, [142].log_data[15].time := 3600.0, [142].log_data[15].valid := 1, [142].log_data[16].time := 3600.0, [142].log_data[16].valid := 1, [142].log_data[17].min := 1.0, [142].log_data[17].max := 1.0, [142].log_data[17].total := 3600.0, [142].log_data[17].time := 3600.0, [142].log_data[17].valid := 1, [142].log_data[18].time := 3600.0, [142].log_data[18].valid := 1,
        [142].log_data[19].time := 3600.0, [142].log_data[19].valid := 1, [142].log_data[20].time := 3600.0, [142].log_data[20].valid := 1, [142].log_data[21].min := 1.0, [142].log_data[21].max := 1.0, [142].log_data[21].total := 3600.0, [142].log_data[21].time := 3600.0, [142].log_data[21].valid := 1, [142].log_data[22].time := 3600.0, [142].log_data[22].valid := 1, [142].log_data[23].time := 3600.0, [142].log_data[23].valid := 1, [142].log_data[24].time := 3600.0, [142].log_data[24].valid := 1, [142].log_data[25].time := 3600.0, [142].log_data[25].valid := 1, [142].log_data[26].time := 3600.0, [142].log_data[26].valid := 1, [142].log_data[27].time := 3600.0, [142].log_data[27].valid := 1, [142].log_data[28].time := 3600.0, [142].log_data[28].valid := 1, [142].log_data[29].min := 1.0, [142].log_data[29].max := 1.0, [142].log_data[29].total := 3600.0, [142].log_data[29].time := 3600.0, [142].log_data[29].valid := 1, [142].log_data[30].min := 1.0, [142].log_data[30].max := 1.0, [142].log_data[30].total := 3600.0, [142].log_data[30].time := 3600.0, [142].log_data[30].valid := 1, [142].log_data[31].max := 1.0, [142].log_data[31].total := 1629.7471, [142].log_data[31].time := 3600.0, [142].log_data[31].maxminute := 8, [142].log_data[31].valid := 1, [142].log_data[32].max := 1.0, [142].log_data[32].total := 1505.749, [142].log_data[32].time := 3600.0, [142].log_data[32].minminute := 6, [142].log_data[32].valid := 1, [142].log_data[33].time := 3600.0, [142].log_data[33].valid := 1, [142].log_data[34].time := 3600.0, [142].log_data[34].valid := 1, [142].log_data[35].max := 1.0, [142].log_data[35].total := 1629.498, [142].log_data[35].time := 3600.0, [142].log_data[35].maxminute := 3, [142].log_data[35].valid := 1, [142].log_data[36].max := 1.0, [142].log_data[36].total := 1440.998, [142].log_data[36].time := 3600.0, [142].log_data[36].minminute := 2, [142].log_data[36].valid := 1, [142].log_data[37].max := 7.5053306, [142].log_data[37].total := 3446.6523, [142].log_data[37].time := 3600.0,
        [142].log_data[37].maxminute := 14, [142].log_data[37].valid := 1, [142].log_data[38].time := 3600.0, [142].log_data[38].valid := 1, [142].log_data[39].min := 0.9947063, [142].log_data[39].max := 1.0210879, [142].log_data[39].total := 3606.9028, [142].log_data[39].time := 3600.0, [142].log_data[39].minminute := 10, [142].log_data[39].maxminute := 16, [142].log_data[39].valid := 1, [142].log_data[40].min := 7.5885, [142].log_data[40].max := 7.630545, [142].log_data[40].total := 27397.697, [142].log_data[40].time := 3600.0, [142].log_data[40].minminute := 28, [142].log_data[40].maxminute := 45, [142].log_data[40].valid := 1, [142].log_data[41].min := 0.02273633, [142].log_data[41].max := 0.023128908, [142].log_data[41].total := 82.556046, [142].log_data[41].time := 3600.0, [142].log_data[41].valid := 1, [142].log_data[42].min := 2.2907004, [142].log_data[42].max := 2.2958827, [142].log_data[42].total := 8257.838, [142].log_data[42].time := 3600.0, [142].log_data[42].minminute := 41, [142].log_data[42].maxminute := 16, [142].log_data[42].valid := 1, [142].log_data[43].min := -0.27999878, [142].log_data[43].max := -0.26000214, [142].log_data[43].total := -1007.67126, [142].log_data[43].time := 3600.0, [142].log_data[43].valid := 1, [142].log_data[44].min := -0.3199997, [142].log_data[44].max := -0.30000305, [142].log_data[44].total := -1090.2708, [142].log_data[44].time := 3600.0, [142].log_data[44].valid := 1, [142].log_data[45].time := 3600.0, [142].log_data[45].valid := 1, [142].log_data[46].time := 3600.0, [142].log_data[46].valid := 1, [142].log_data[47].time := 3600.0, [142].log_data[47].valid := 1, [142].log_data[48].min := 6.587924, [142].log_data[48].max := 6.9465485, [142].log_data[48].total := 24232.408, [142].log_data[48].time := 3600.0, [142].log_data[48].minminute := 45, [142].log_data[48].maxminute := 18, [142].log_data[48].valid := 1, [142].log_data[49].min := 6.8263917, [142].log_data[49].max := 9.640621, [142].log_data[49].total := 29813.418, [142].log_data[49].time := 3600.0, [142].log_data[49].minminute := 42, [142].log_data[49].maxminute := 11, [142].log_data[49].valid := 1,
